// TwinCAT 3 PLC project Xts_Library
// Title: Xts Library
// Company: BeckhoffUK
// Author: ChrisK
// ProjectVersion: 7.2.0.0
// Description: Xts framework implementation
// ProgramVersion: 3.1.4026.13
// libraries:
//   Base Library, * (Beckhoff UK)
//   Motion Library, * (Beckhoff UK)
//   Tc2_MC2, * (Beckhoff Automation GmbH)
//   Tc2_Standard, * (Beckhoff Automation GmbH)
//   Tc2_System, * (Beckhoff Automation GmbH)
//   Tc3_Mc3Definitions, * (Beckhoff Automation GmbH)
//   Tc3_McCollisionAvoidance, * (Beckhoff Automation GmbH)
//   Tc3_McCoordinatedMotion, * (Beckhoff Automation GmbH)
//   Tc3_Module, * (Beckhoff Automation GmbH)
//   Tc3_PackML_V2, * (Beckhoff Automation GmbH)
//   Tc3_XTS_Utility, * (Beckhoff Automation GmbH)
// project tree:
//   Mover Class/ ITF_XtsMoverAxis.TcIO, XtsMoverAxis.TcPOU
//   SequenceSamples/ IndexMoverSequence.TcPOU, IndexSequenceState.TcDUT, MoverSequenceInfo.TcDUT
//   Station Class/Process/ IProcess.TcIO, Process.TcPOU
//   Station Class/Station/ IStation.TcIO, Station.TcPOU, StationSample.TcPOU, stStationInfo.TcDUT, stStationStatus.TcDUT
//   Station Class/TMSStation/ ITF_SwitchStation.TcIO, TmsEmbarkSingleSwitch.TcPOU, TmsEmbarkStation.TcPOU, TmsHoldStation.TcPOU
//   / SystemParameters.TcGVL
//   Tasks/ ActivateTrackForMover.TcPOU, AddMoverToGroupTask.TcPOU, DisableGroup.TcPOU, EnableGroup.TcPOU, GearInCA.TcPOU, HaltMover.TcPOU, MoveModuloMoverToPosition.TcPOU, RemoveAllMoverFromGroup.TcPOU, RemoveMoverFromGroup.TcPOU, ResetGroup.TcPOU, StopMoverGroup.TcPOU, XtsDisableSequence.TcPOU, XtsEnableSequence.TcPOU
//   XTS Class/XPU/ ITF_XTSIOEnvVarWrapper.TcIO, XTSIOEnvVarWrapper.TcPOU
//   XTS Class/Xts Collision Group/ CAGroupInfo.TcDUT, CAGroupStatus.TcDUT, CollisionGroup.TcPOU, ICollisionGroup.TcIO, ITF_CAMover.TcIO
//   XTS Class/Xts Hardware/ I_XtsTrack.TcIO, XtsSystemInitialisation.TcDUT, XTSHardware_V2.TcPOU, XtsMotorModule.TcPOU, XtsPart.TcPOU, XtsTrack.TcPOU
//   XTS Class/ Xts.TcPOU
// real-time tasks:
//   TASK PlcTask: cycle T#10ms, priority 20, ADS port 350

// ---- SequenceSamples/IndexSequenceState.TcDUT
{attribute 'qualified_only'}
{attribute 'strict'}
TYPE IndexSequenceState :
(
	Init := 0,                                               
	Available := 1,
	MovingToStart := 2, 
	AtStart := 3,                                 
	MovingToStation := 4,
	QueuedAtStation := 5,
	AtStation := 6,
	AtProcess := 7,
	InProcess := 8,
	GetNextMove := 9,
	GoToNextStation := 10,
	Stopping := 11,
	Aborting := 12
);
END_TYPE

// ---- SequenceSamples/MoverSequenceInfo.TcDUT
TYPE MoverSequenceInfo :
STRUCT
	MoverId : UDINT;
	CurrentStation : INT;
	Velocity : MC_LREAL;
	State : IndexSequenceState;
END_STRUCT
END_TYPE

// ---- Station Class/Station/stStationInfo.TcDUT
TYPE stStationInfo :
STRUCT
	StationProcessTime : TIME;
	StationPosition : MC_LREAL;
	StationStatus : stStationStatus;
END_STRUCT
END_TYPE

// ---- Station Class/Station/stStationStatus.TcDUT
TYPE stStationStatus :
STRUCT
	Empty : BOOL;
	Complete : BOOL;
	Operating : BOOL;
	Ready : BOOL;
	HasMover : BOOL;
END_STRUCT
END_TYPE

// ---- XTS Class/Xts Collision Group/CAGroupInfo.TcDUT
TYPE CAGroupInfo :
STRUCT
	sName 		: STRING;
	nId			: OTCID;
	eGroupState	: MC_GROUP_STATE;
	nAxesCount 	: INT; 
END_STRUCT
END_TYPE

// ---- XTS Class/Xts Collision Group/CAGroupStatus.TcDUT
{attribute 'qualified_only'}
{attribute 'strict'}
TYPE CAGroupStatus :
(
	mcGroupStateInvalid:=0, 
	mcGroupStateDisabled:=1,
	mcGroupStateStandby:=2, 
	mcGroupStateMoving:=3, 
	mcGroupStateStopping:=4, 
	mcGroupStateErrorStop:=5, 
	mcGroupStateHoming:=6, 
	mcGroupStateNotReady:=7, 
	mcGroupAllAxesStanding:=8,
    mcGroupConstantVelocity:=9,
    mcGroupAccelerating:=10,
    mcGroupDecelerating:=11,
    mcGroupInPosition:=12,
    mcGroupError:=13
);
END_TYPE

// ---- XTS Class/Xts Hardware/XtsSystemInitialisation.TcDUT
{attribute 'qualified_only'}
{attribute 'strict'}
TYPE XtsSystemInitialisation :
(
	Init := 0,
	PassGroupReference := 1,
	InitialiseHardware := 2,
	SetDetection := 3,                                              
	Redetect := 4,
	MoversValid := 5,                                 
	AllMoversFound := 6,
	MoverIdDetection := 7,
	XTSMode := 8,
	CheckModuleVoltages := 9,
	HWReady := 10,
	HWError := 999
);
END_TYPE

// ---- SystemParameters.TcGVL
{attribute 'qualified_only'}
VAR_GLOBAL CONSTANT
	MaxModulesInPart  : UINT := 20;
	MaxPartsInTrack : UINT := 5;
	NumberOfMovers : UINT := 10;
	NumberOfStations : UINT := 6;
	NumberOfParts : UINT := 1;
	NumberOfTracks : UINT := 2;
END_VAR

// ---- Mover Class/ITF_XtsMoverAxis.TcIO
INTERFACE ITF_XtsMoverAxis

PROPERTY Acceleration : mc_lreal
GET
END_GET
SET
END_SET
END_PROPERTY

METHOD ActivateTrack : HRESULT
VAR_INPUT
	NewTrack : OTCID;
	Track : I_XtsTrack;
END_VAR
END_METHOD

PROPERTY AxisRef : Reference to Axis_ref
GET
END_GET
END_PROPERTY

PROPERTY Deceleration : mc_lreal
GET
END_GET
SET
END_SET
END_PROPERTY

METHOD DisableMover : HRESULT
VAR_INPUT
END_VAR
END_METHOD

METHOD EnableMover : HRESULT
VAR_INPUT
END_VAR
END_METHOD

PROPERTY Gap : MC_LREAL
GET
END_GET
SET
END_SET
END_PROPERTY

METHOD PUBLIC Gear : HRESULT
VAR_INPUT
	MasterPosition : MC_LREAL;
	SlavePosition : MC_LREAL;
END_VAR
END_METHOD

METHOD HaltAxis : HRESULT
VAR_INPUT
END_VAR
END_METHOD

PROPERTY PUBLIC IdentInGroup : IDENT_IN_GROUP_REF
GET
END_GET
END_PROPERTY

METHOD isMoverAtPosition : BOOL
VAR_INPUT
	Position : MC_LREAL;
END_VAR
END_METHOD

METHOD isMoverDetected : BOOL
VAR_INPUT
END_VAR
END_METHOD

METHOD isMoverEnabled : BOOL
VAR_INPUT
END_VAR
END_METHOD

METHOD isMoverStationary : BOOL
VAR_INPUT
END_VAR
END_METHOD

PROPERTY Jerk : mc_lreal
GET
END_GET
SET
END_SET
END_PROPERTY

PROPERTY PUBLIC MoverErrorID : DWORD
GET
END_GET
END_PROPERTY

PROPERTY PUBLIC MoversActiveTrack : OTCID
GET
END_GET
END_PROPERTY

PROPERTY PUBLIC MoverXtsIoEnvInterface : I_TcIoXtsXpuMover
GET
END_GET
SET
END_SET
END_PROPERTY

METHOD MoveTo : HRESULT
VAR_INPUT
	RequiredPosition : MC_LREAL;
	MoveVelocity : MC_LREAL;
	NonModuloMove : BOOL;
END_VAR
END_METHOD

PROPERTY MyCAGroup : ITF_CAMover
GET
END_GET
SET
END_SET
END_PROPERTY

PROPERTY MyMasterRef : REFERENCE TO AXIS_REF
GET
END_GET
SET
END_SET
END_PROPERTY

PROPERTY PositiveDirectionOnly : BOOL
GET
END_GET
SET
END_SET
END_PROPERTY

METHOD ResetAxis : HRESULT
VAR_INPUT
END_VAR
END_METHOD

METHOD TriggerMoverArrive : BOOL
VAR_INPUT
END_VAR
END_METHOD

METHOD TriggerMoverLeave : BOOL
VAR_INPUT
END_VAR
END_METHOD

END_INTERFACE

// ---- Station Class/Process/IProcess.TcIO
INTERFACE IProcess EXTENDS IStation

PROPERTY EndPosition : MC_LREAL
GET
END_GET
SET
END_SET
END_PROPERTY

PROPERTY IsProcess : booL
GET
END_GET
SET
END_SET
END_PROPERTY

PROPERTY ProcessVelocity : mc_lreal
GET
END_GET
SET
END_SET
END_PROPERTY

PROPERTY StartPosition : MC_LREAL
GET
END_GET
SET
END_SET
END_PROPERTY

END_INTERFACE

// ---- Station Class/Station/IStation.TcIO
INTERFACE IStation

METHOD Abort : BOOL
VAR_INPUT
END_VAR
END_METHOD

METHOD HasMover : BOOL
VAR_INPUT
	mover : ITF_XtsMoverAxis;
END_VAR
END_METHOD

METHOD IsClear : BOOL
VAR_INPUT
END_VAR
END_METHOD

METHOD isComplete : BOOL
VAR_INPUT
END_VAR
END_METHOD

PROPERTY IsLastStation : BOOL
GET
END_GET
SET
END_SET
END_PROPERTY

METHOD IsOperating : BOOL
VAR_INPUT
END_VAR
END_METHOD

METHOD IsReady : BOOL
VAR_INPUT
END_VAR
END_METHOD

METHOD MoverAway : BOOL
VAR_INPUT
END_VAR
END_METHOD

PROPERTY Position : MC_LREAL
GET
END_GET
SET
END_SET
END_PROPERTY

END_INTERFACE

// ---- Station Class/TMSStation/ITF_SwitchStation.TcIO
INTERFACE ITF_SwitchStation EXTENDS __SYSTEM.IQueryInterface

METHOD SwitchMoveComplete : BOOL
VAR_INPUT
END_VAR
END_METHOD

END_INTERFACE

// ---- XTS Class/XPU/ITF_XTSIOEnvVarWrapper.TcIO
INTERFACE ITF_XTSIOEnvVarWrapper

METHOD GetCaGroupInterface : I_Mc2CaGroup
VAR_INPUT
	CAGroupNumber : INT;
END_VAR
END_METHOD

METHOD PUBLIC GetMotorModuleInterface : I_TcIoXtsPartModule
VAR_INPUT
	PartNumber : INT;
	ModuleNumber : INT;
END_VAR
END_METHOD

METHOD PUBLIC GetMoverInterface : I_TcIoXtsXpuMover
VAR_INPUT
	MoverId : INT;
END_VAR
END_METHOD

METHOD PUBLIC GetPartInterface : I_TcIoXtsXpuPart
VAR_INPUT
	PartNumber : INT;
END_VAR
END_METHOD

METHOD PUBLIC GetTrackInterface : I_TcIoXtsXpuTrack
VAR_INPUT
	TrackNumber : INT;
END_VAR
END_METHOD

METHOD GetXPUInterface : I_TcIoXtsProcessingUnit
VAR_INPUT
END_VAR
END_METHOD

METHOD IsInitialised : BOOL
VAR_INPUT
END_VAR
END_METHOD

METHOD IsInSim : BOOL
VAR_INPUT
END_VAR
END_METHOD

END_INTERFACE

// ---- XTS Class/Xts Collision Group/ICollisionGroup.TcIO
INTERFACE ICollisionGroup

METHOD AddMoverToThisGroup : HRESULT
VAR_INPUT
	MoverToAdd : ITF_XtsMoverAxis;
END_VAR
END_METHOD

METHOD Disable : BOOL
VAR_INPUT
END_VAR
END_METHOD

METHOD Enable : BOOL
VAR_INPUT
END_VAR
END_METHOD

METHOD GetAxisCount : udint
VAR_INPUT
END_VAR
END_METHOD

PROPERTY GroupRef : reference to AXES_GROUP_REF
GET
END_GET
END_PROPERTY

PROPERTY GroupState : CAGroupStatus
GET
END_GET
END_PROPERTY

METHOD GroupStop : HRESULT
VAR_INPUT
END_VAR
END_METHOD

METHOD RemoveAllMovers : HRESULT
VAR_INPUT
END_VAR
END_METHOD

METHOD Reset : BOOL
VAR_INPUT
END_VAR
END_METHOD

END_INTERFACE

// ---- XTS Class/Xts Collision Group/ITF_CAMover.TcIO
INTERFACE ITF_CAMover

METHOD AddMoverToThisGroup : HRESULT
VAR_INPUT
	MoverToAdd : ITF_XtsMoverAxis;
END_VAR
END_METHOD

METHOD RemoveAMover : BOOL
VAR_INPUT
	moverId : UDINT;
END_VAR
END_METHOD

END_INTERFACE

// ---- XTS Class/Xts Hardware/I_XtsTrack.TcIO
INTERFACE I_XtsTrack

PROPERTY MyOTCID : OTCID
GET
END_GET
SET
END_SET
END_PROPERTY

PROPERTY TrackLength : MC_Lreal
GET
END_GET
END_PROPERTY

END_INTERFACE

// ---- Mover Class/XtsMoverAxis.TcPOU
FUNCTION_BLOCK XtsMoverAxis EXTENDS CyclicBase IMPLEMENTS ITF_XtsMoverAxis
VAR
	MyAxisRef : AXIS_REF;
	_MyAxisStatus : ST_AxisStatus;
	_MyNCData : NCTOPLC_AXIS_REF;
	MoverPowerCommand : AxisPower(MyAxisRef);
	MoverMoveCommand : MoveModuloMoverToPosition(MyAxisRef) := (Gap := 100.0);
	MoverHaltCommand : HaltMover(MyAxisRef);
	MoverResetCommand : AxesReset(MyAxisRef);
	MoverActivateTrackCommand : ActivateTrackForMover(MyAxisRef);
	axesGear	: GearInCA(MyAxisRef);
	_ipTcIoXtsMover	: I_TcIoXtsXpuMover;
	_ActiveTrackLength : MC_LREAL;
	TrackChangeTrigger : R_TRIG;
	_MoverAbsMoveOptions : ST_MoveAbsoluteCAOptions;
	_stTmsActPositions			: ST_PositionInfo;
	_CurrentTrack : I_XtsTrack;
	_MyCAGroup : ITF_CAMover;
	_ForwardOnly : BOOL := TRUE;
END_VAR
VAR CONSTANT
	_MaxMoverVelocity : MC_LREAL := 4000.0;
END_VAR

PROPERTY PUBLIC Acceleration : MC_LREAL
GET
Acceleration := MoverMoveCommand.Acceleration;
END_GET
SET
MoverMoveCommand.Acceleration := Acceleration;
END_SET
END_PROPERTY

METHOD ActivateTrack : HRESULT
VAR_INPUT
	NewTrack : OTCID;
	Track : I_XtsTrack;
END_VAR
IF NOT MoverActivateTrackCommand.Busy AND THIS^.isMoverStationary() AND NewTrack <> 0  THEN
	IF MoverActivateTrackCommand.Execute(Track := Track.MyOTCID) THEN
		_CurrentTrack := Track;
		_ActiveTrackLength := Track.TrackLength;
		ActivateTrack := 1;
	ELSE
		ActivateTrack := -1;
	END_IF
ELSE
	ActivateTrack := -1;
END_IF
END_METHOD

METHOD ActivateZeroReferenceSystem : HRESULT
VAR_INPUT
	NewTrack : OTCID;
END_VAR
IF NOT MoverActivateTrackCommand.Busy AND THIS^.isMoverStationary() THEN // AND NewTrack <> 0  THEN
	IF MoverActivateTrackCommand.Execute(Track := NewTrack) THEN
		_CurrentTrack := 0;
		ActivateZeroReferenceSystem := 1;
	ELSE
		ActivateZeroReferenceSystem := -1;
	END_IF
ELSE
	ActivateZeroReferenceSystem := -1;
END_IF
END_METHOD

PROPERTY AxisRef : Reference to Axis_ref
GET
AxisRef REF= MyAxisRef;
END_GET
END_PROPERTY

METHOD PUBLIC  Cycle : HRESULT
VAR_INPUT
END_VAR
IF isMoverDetected() THEN
	MoverPowerCommand.Cycle();
	MoverMoveCommand.Cycle();
	MoverHaltCommand.Cycle();
	MoverResetCommand.Cycle();
	MoverActivateTrackCommand.Cycle();
	axesGear.Cycle();
	TrackChangeTrigger(CLK := MoverActivateTrackCommand.Done);
	IF TrackChangeTrigger.Q THEN
		_MoverAbsMoveOptions.PositionReferenceSystem :=  MoverActivateTrackCommand.NewTrackId;
		_MoverAbsMoveOptions.DynamicsReferenceSystem := MoverActivateTrackCommand.NewTrackId;
		MoverMoveCommand.Options := _MoverAbsMoveOptions;	
	END_IF
	IF _ipTcIoXtsMover <> 0 THEN
		_stTmsActPositions := _ipTcIoXtsMover.GetPositionInfo();
	END_IF
	Cycle := 1;
ELSE
	Cycle := -1;
END_IF
MyAxisRef.ReadStatus();
_MyNCData := MyAxisRef.NcToPlc;
_MyAxisStatus := MyAxisRef.Status;
END_METHOD

PROPERTY PUBLIC Deceleration : MC_LREAL
GET
Deceleration := MoverMoveCommand.Deceleration;
END_GET
SET
MoverMoveCommand.Deceleration := Deceleration;
MoverHaltCommand.Deceleration := Deceleration;
END_SET
END_PROPERTY

METHOD PUBLIC DisableMover : HRESULT
VAR_INPUT
END_VAR
IF THIS^.isMoverEnabled() AND NOT MoverPowerCommand.Busy THEN
	MoverPowerCommand.Disable();
	DisableMover := 1;
ELSE
	DisableMover := -1;
END_IF
END_METHOD

METHOD PUBLIC EnableMover : HRESULT
VAR_INPUT
END_VAR
IF (NOT MoverPowerCommand.Busy) AND NOT THIS^.isMoverEnabled() THEN // AND _CurrentTrack <> 0 THEN
	MoverPowerCommand.Enable();
	EnableMover := 1;
ELSE
	EnableMover := -1;
END_IF
END_METHOD

PROPERTY PUBLIC Gap : MC_LREAL
GET
Gap := MoverMoveCommand.Gap;
END_GET
SET
IF Gap >= 50.0 THEN
	MoverMoveCommand.Gap := Gap;
	MoverHaltCommand.Gap := Gap;
ELSE
	Gap := 100.0;
END_IF
END_SET
END_PROPERTY

METHOD PUBLIC Gear : HRESULT
VAR_INPUT
	MasterPosition : MC_LREAL;
	SlavePosition : MC_LREAL;
END_VAR
IF NOT axesGear.Busy AND __ISVALIDREF(axesGear.MyGearMaster) AND MasterPosition <= _ActiveTrackLength AND SlavePosition <= _ActiveTrackLength THEN
	IF axesGear.Sync(MasterPosition := MasterPosition, SlavePosition := SlavePosition) THEN
		Gear := 1;
	ELSE
		Gear := -1;
	END_IF
ELSE
	Gear := -1;
END_IF
END_METHOD

METHOD GetMoverCtrlOTCID : XtsMoverControllerOTCID
VAR_INPUT
END_VAR
GetMoverCtrlOTCID := _ipTcIoXtsMover.P_MoverControllerOid;
END_METHOD

METHOD GetMoverOTCID : OTCID
VAR_INPUT
END_VAR
//GetMoverCtrlOTCID := _ipTcIoXtsMover.P_AxisOid;
END_METHOD

METHOD PUBLIC HaltAxis : HRESULT
VAR_INPUT
END_VAR
IF NOT MoverHaltCommand.Busy THEN// AND NOT THIS^.isMoverStationary() THEN
	IF MoverHaltCommand.Execute() THEN
		HaltAxis := 1;
	ELSE
		HaltAxis := -1;
	END_IF
ELSE
	HaltAxis := -1;
END_IF
END_METHOD

PROPERTY PUBLIC IdentInGroup : IDENT_IN_GROUP_REF
GET
IdentInGroup := UDINT_TO_IDENTINGROUP(id := _MyNCData.AxisId);
END_GET
END_PROPERTY

METHOD inGear : BOOL
VAR_INPUT
END_VAR
inGear := axesGear.GearInPosCA.InSync;
END_METHOD

METHOD IsActive : BOOL
VAR_INPUT
END_VAR
IsActive := _ipTcIoXtsMover.GetIsActive();
END_METHOD

METHOD PUBLIC isMoverAtPosition : BOOL
VAR_INPUT
	Position : MC_LREAL;
END_VAR
IF Position > 1 THEN
	IF _stTmsActPositions.fTrackPosition < position + 1 AND _stTmsActPositions.fTrackPosition > position - 1 THEN
		isMoverAtPosition := TRUE;
	ELSE
		isMoverAtPosition := FALSE;
	END_IF  
ELSE
	IF _stTmsActPositions.fTrackPosition < position + 1 AND _stTmsActPositions.fTrackPosition > 0.0  
		OR _stTmsActPositions.fTrackPosition < _CurrentTrack.TrackLength AND _stTmsActPositions.fTrackPosition > _CurrentTrack.TrackLength - 1 THEN
		isMoverAtPosition := TRUE;
	ELSE
		isMoverAtPosition := FALSE;
	END_IF
END_IF
END_METHOD

METHOD PUBLIC isMoverDetected : BOOL
VAR_INPUT
END_VAR
isMoverDetected := _MyNCData.AxisId <> 0;
END_METHOD

METHOD PUBLIC isMoverEnabled : BOOL
VAR_INPUT
END_VAR
isMoverEnabled :=  NOT _MyAxisStatus.Disabled;
END_METHOD

METHOD PUBLIC isMoverStationary : BOOL
VAR_INPUT
END_VAR
isMoverStationary := _MyAxisStatus.NotMoving;
END_METHOD

PROPERTY PUBLIC Jerk : MC_LREAL
GET
Jerk := MoverMoveCommand.Jerk;
END_GET
SET
MoverMoveCommand.Jerk := Jerk;
MoverHaltCommand.Jerk := Jerk;
END_SET
END_PROPERTY

PROPERTY PUBLIC MoverErrorID : DWORD
GET
MoverErrorID := _MyAxisStatus.ErrorID;
END_GET
END_PROPERTY

PROPERTY PUBLIC MoversActiveTrack : OTCID
GET
MoversActiveTrack := _ipTcIoXtsMover.GetActiveTrackObjectId();
END_GET
END_PROPERTY

PROPERTY PUBLIC MoverXtsIoEnvInterface : I_TcIoXtsXpuMover
GET
MoverXtsIoEnvInterface := _ipTcIoXtsMover;
END_GET
SET
_ipTcIoXtsMover := MoverXtsIoEnvInterface;
END_SET
END_PROPERTY

METHOD PUBLIC MoveTo : HRESULT
VAR_INPUT
	RequiredPosition : MC_LREAL;
	MoveVelocity : MC_LREAL;
	NonModuloMove : BOOL;
END_VAR
IF NOT MoverMoveCommand.Busy AND MoveVelocity < _MaxMoverVelocity AND (*RequiredPosition < _ActiveTrackLength AND*) Gap >= 50.0 THEN
	IF NonModuloMove THEN
		IF THIS^.MoverMoveCommand.MoveTo(Position := RequiredPosition, 
										Velocity := MoveVelocity, 
										Direction := Tc3_Mc3Definitions.MC_DIRECTION.mcDirectionNonModulo, 
										Turns := 0) THEN
										
			MoveTo := 1;
		END_IF
	ELSE
		IF _ForwardOnly THEN
			THIS^.MoverMoveCommand.MoveTo(Position := RequiredPosition, 
										Velocity := MoveVelocity, 
										Direction := Tc3_Mc3Definitions.MC_DIRECTION.mcDirectionPositive, 
										Turns := 0);
			MoveTo := 1;
		ELSE
			IF RequiredPosition > MyAxisRef.NcToPlc.ModuloActPos THEN
				IF THIS^.MoverMoveCommand.MoveTo(Position := RequiredPosition, 
											Velocity := MoveVelocity, 
											Direction := Tc3_Mc3Definitions.MC_DIRECTION.mcDirectionPositive, 
											Turns := 0) THEN
											
					MoveTo := 1;
				END_IF
			ELSE
				IF THIS^.MoverMoveCommand.MoveTo(Position := RequiredPosition, 
											Velocity := MoveVelocity, 
											Direction := Tc3_Mc3Definitions.MC_DIRECTION.mcDirectionNegative, 
											Turns := 0) THEN
											
					MoveTo := 1;
				END_IF	
			END_IF
		END_IF
	END_IF
ELSE
	MoveTo := -1;
END_IF
END_METHOD

PROPERTY MyCAGroup : ITF_CAMover
GET
MyCAGroup := _MyCAGroup;
END_GET
SET
_MyCAGroup := MyCAGroup;
END_SET
END_PROPERTY

PROPERTY MyMasterRef : REFERENCE TO AXIS_REF
GET
MyMasterRef REF= axesGear.MyGearMaster;
END_GET
SET
axesGear.MyGearMaster REF= MyMasterRef;
END_SET
END_PROPERTY

PROPERTY PositiveDirectionOnly : BOOL
GET
PositiveDirectionOnly := _ForwardOnly;
END_GET
SET
_ForwardOnly := PositiveDirectionOnly;
END_SET
END_PROPERTY

METHOD PUBLIC ResetAxis : HRESULT
VAR_INPUT
END_VAR
IF NOT MoverResetCommand.Busy AND _MyAxisStatus.Error THEN
	IF MoverResetCommand.Execute() = S_OK THEN
		ResetAxis := 1;
	ELSE
		ResetAxis := -1;
	END_IF
ELSE
	ResetAxis := -1;
END_IF
END_METHOD

METHOD SetForceCouple : HRESULT
VAR_INPUT
	XtsMoverCtrlOTCID : Tc3_XTS_Utility.XtsMoverControllerOTCID;
END_VAR
_ipTcIoXtsMover.MoverController.SetForceCouple(nForceCouple := XtsMoverCtrlOTCID);
END_METHOD

METHOD SwapMover : HRESULT
VAR_INPUT
    MoverToSwapWith : MoverOTCID;
END_VAR
_ipTcIoXtsMover.swapmover(nSwapMoverObjectId := MoverToSwapWith);
END_METHOD

METHOD TriggerMoverArrive : BOOL
VAR_INPUT
END_VAR
_ipTcIoXtsMover.TriggerArrive();
END_METHOD

METHOD TriggerMoverLeave : BOOL
VAR_INPUT
END_VAR
TriggerMoverLeave := _ipTcIoXtsMover.TriggerLeave();
END_METHOD

END_FUNCTION_BLOCK

// ---- Tasks/MoveModuloMoverToPosition.TcPOU
FUNCTION_BLOCK MoveModuloMoverToPosition EXTENDS TaskBase
VAR_INPUT
END_VAR
VAR_OUTPUT
END_VAR
VAR
	moveAbs	: MC_MoveAbsoluteCA;
	_Axis : REFERENCE TO AXIS_REF;
	_MoveMover : BOOL;
	_stOptions : ST_MoveAbsoluteCAOptions;
	_ErrorId: UDINT;
END_VAR

{analysis -2}

METHOD Abort : BOOL
moveAbs.Execute := FALSE;
moveAbs.Position := moveAbs.Velocity := 0;
_MoveMover := false;
_Busy := FALSE;
Abort := true;
State := 0;
END_METHOD

PROPERTY PUBLIC Acceleration : mc_lreal
GET
Acceleration := moveAbs.Acceleration;
END_GET
SET
moveAbs.Acceleration := Acceleration;
END_SET
END_PROPERTY

METHOD Cycle : HRESULT
VAR_INPUT
END_VAR
Cycle := S_OK;
CASE State OF
	0:
		IF _MoveMover THEN
			Cycle := S_PENDING;
			_Done := FALSE;
			_Error := FALSE;
			_Busy := TRUE;
			moveAbs.Execute := TRUE;
			IF moveAbs.Busy THEN
				State := 10;
				_MoveMover := FALSE;
			END_IF
		END_IF
		
	10:
		IF NOT moveAbs.Busy THEN
			IF moveAbs.Done THEN
				_Done := TRUE;
			ELSIF moveAbs.Error THEN
				_Error := TRUE;
				_ErrorId := moveAbs.ErrorId;
			END_IF
			_Busy := FALSE;
			moveAbs.Execute := FALSE;
			State := 0;
			Cycle := S_OK;
		END_IF
	ELSE
		Cycle := E_FAIL;
END_CASE

moveAbs(Axis := _Axis, Options := _stOptions);
END_METHOD

PROPERTY PUBLIC Deceleration : mc_lreal
GET
Deceleration := moveAbs.Deceleration;
END_GET
SET
moveAbs.Deceleration := Deceleration;
END_SET
END_PROPERTY

METHOD FB_init : BOOL
VAR_INPUT
	bInitRetains : BOOL; // if TRUE, the retain variables are initialized (warm start / cold start)
	bInCopyCode : BOOL;  // if TRUE, the instance afterwards gets moved into the copy code (online change)
	axis : reference TO AXIS_REF;
END_VAR
_Axis REF= axis;
END_METHOD

PROPERTY PUBLIC Gap : mc_lreal
GET
Gap := moveAbs.Gap;
END_GET
SET
moveAbs.Gap := Gap;
END_SET
END_PROPERTY

PROPERTY PUBLIC Jerk : mc_lreal
GET
Jerk := moveAbs.Jerk;
END_GET
SET
moveAbs.Jerk := Jerk;
END_SET
END_PROPERTY

METHOD MoveTo : BOOL
VAR_INPUT
	Position : MC_LREAL;
	Velocity : MC_LREAL;
	Direction: Tc3_Mc3Definitions.MC_DIRECTION;
	Turns: UDINT;
END_VAR
moveAbs.Position := Position;
moveAbs.Velocity := Velocity;
moveAbs.Direction := Direction;
moveAbs.Options.AdditionalTurns := Turns;
_MoveMover := MoveTo := true;
END_METHOD

PROPERTY PUBLIC Options : ST_MoveAbsoluteCAOptions
GET
Options := _stOptions;
END_GET
SET
_stOptions := Options;
END_SET
END_PROPERTY

END_FUNCTION_BLOCK

// ---- Tasks/HaltMover.TcPOU
FUNCTION_BLOCK HaltMover EXTENDS TaskBase
VAR_INPUT
END_VAR
VAR_OUTPUT
END_VAR
VAR
	haltMoverCA : Tc3_McCollisionAvoidance.MC_HaltCA;
	_Axis : REFERENCE TO Tc2_MC2.AXIS_REF;
	_HaltMover : BOOL;
END_VAR

{analysis -2}

METHOD Abort : BOOL
haltMoverCA.Execute := FALSE;
_Busy := FALSE;
_HaltMover := FALSE;
Abort := TRUE;
State := 0;
END_METHOD

METHOD Cycle : HRESULT
VAR_INPUT
END_VAR
Cycle := S_OK;
CASE State OF
	0:
		IF _HaltMover THEN
			Cycle := S_PENDING;
			_Done := FALSE;
			_Error := FALSE;
			_Busy := TRUE;
			haltMoverCA.Execute := TRUE;
			IF haltMoverCA.Busy THEN
				State := 10;
				_HaltMover := FALSE;
			END_IF
		END_IF
	
	10:
		IF NOT haltMoverCA.Busy THEN
			IF haltMoverCA.Done THEN
				_Done := TRUE;
			ELSIF haltMoverCA.Error THEN
				_Error := TRUE;
			END_IF
			_Busy := FALSE;
			haltMoverCA.Execute := FALSE;
			State := 0;
			Cycle := S_OK;
		END_IF
	ELSE
		Cycle := E_FAIL;
END_CASE

haltMoverCA(Axis := _Axis);
END_METHOD

PROPERTY Deceleration : MC_LREAL
GET
Deceleration := haltMoverCA.Deceleration;
END_GET
SET
haltMoverCA.Deceleration := Deceleration;
END_SET
END_PROPERTY

METHOD Execute : BOOL
VAR_INPUT
END_VAR
IF NOT _HaltMover THEN
	Execute := _HaltMover := TRUE;
ELSE
	Execute := false;
END_IF
END_METHOD

METHOD FB_init : BOOL
VAR_INPUT
	bInitRetains : BOOL; // if TRUE, the retain variables are initialized (warm start / cold start)
	bInCopyCode : BOOL;  // if TRUE, the instance afterwards gets moved into the copy code (online change)
	Axis : reference TO AXIS_REF;
END_VAR
_Axis REF= Axis;
END_METHOD

PROPERTY Gap : MC_LREAL
GET
Gap := haltMoverCA.Gap;
END_GET
SET
haltMoverCA.Gap := Gap;
END_SET
END_PROPERTY

PROPERTY Jerk : MC_LREAL
GET
Jerk := haltMoverCA.Jerk;
END_GET
SET
haltMoverCA.Jerk := Jerk;
END_SET
END_PROPERTY

END_FUNCTION_BLOCK

// ---- Tasks/ActivateTrackForMover.TcPOU
FUNCTION_BLOCK ActivateTrackForMover EXTENDS TaskBase
VAR_INPUT
END_VAR
VAR_OUTPUT
END_VAR
VAR
	mcActivateTrack : Tc3_McCollisionAvoidance.MC_ActivateTrack;
	_Axis : REFERENCE TO Tc2_MC2.AXIS_REF;
	_ActivateTrack : BOOL;
	_newTrackId : OTCID;
	_errorId: UDINT;
END_VAR

{analysis -2}

METHOD Abort : BOOL
mcActivateTrack.Execute := FALSE;
_Busy := FALSE;
_ActivateTrack := FALSE;
Abort := TRUE;
State := 0;
END_METHOD

METHOD Cycle : HRESULT
VAR_INPUT
END_VAR
Cycle := S_OK;
CASE State OF
	0:
		IF _ActivateTrack THEN
			Cycle := S_PENDING;
			_Done := FALSE;
			_Error := FALSE;
			_Busy := TRUE;
			mcActivateTrack.Execute := TRUE;
			IF mcActivateTrack.Busy THEN
				State := 10;
				_ActivateTrack := FALSE;
			END_IF
		END_IF
	
	10:
		IF NOT mcActivateTrack.Busy THEN
			IF mcActivateTrack.Done THEN
				_Done := TRUE;
				_newTrackId := mcActivateTrack.TrackId;
			ELSIF mcActivateTrack.Error THEN
				_Error := TRUE;
				_errorId := mcActivateTrack.ErrorId;
			END_IF
			_Busy := FALSE;
			mcActivateTrack.Execute := FALSE;
			State := 0;
			Cycle := S_OK;
		END_IF
	ELSE
		Cycle := E_FAIL;
END_CASE

mcActivateTrack(Axis := _Axis);
END_METHOD

METHOD PUBLIC Execute : BOOL
VAR_INPUT
	Track : OTCID;
END_VAR
IF NOT _ActivateTrack THEN
	Execute := _ActivateTrack := TRUE;
	mcActivateTrack.TrackId := Track;
ELSE
	Execute := false;
END_IF;
END_METHOD

METHOD FB_init : BOOL
VAR_INPUT
	bInitRetains : BOOL; // if TRUE, the retain variables are initialized (warm start / cold start)
	bInCopyCode : BOOL;  // if TRUE, the instance afterwards gets moved into the copy code (online change)
	Axis : reference TO AXIS_REF;
END_VAR
_Axis REF= Axis;
END_METHOD

PROPERTY PUBLIC NewTrackId : OTCID
GET
NewTrackId := _newTrackId;
END_GET
END_PROPERTY

END_FUNCTION_BLOCK

// ---- Tasks/GearInCA.TcPOU
FUNCTION_BLOCK PUBLIC GearInCA EXTENDS TaskBase
VAR
	GearInPosCA : Tc3_McCollisionAvoidance.MC_GearInPosCA;
	_syncStrategy : Tc3_Mc3Definitions.MC_SYNC_STRATEGY := Tc3_Mc3Definitions.MC_SYNC_STRATEGY.mcSyncStrategyEarly;
	_SlaveAxis : REFERENCE TO Tc2_MC2.AXIS_REF;
	_MasterAxis : REFERENCE TO Tc2_MC2.AXIS_REF;
	_GearMover: BOOL;
	_ErrorID: UDINT;
END_VAR

{analysis -2}

METHOD Abort : BOOL
GearInPosCA.Execute := FALSE;
_GearMover := FALSE;
_Busy := false;
Abort := true;
State := 0;
END_METHOD

METHOD Cycle : HRESULT
VAR_INPUT
END_VAR
Cycle := S_OK;
CASE State OF
	0:
		IF _GearMover THEN
			Cycle := S_PENDING;
			_Done := FALSE;
			_Error := FALSE;
			_Busy := TRUE;
			GearInPosCA.Execute := TRUE;
			IF GearInPosCA.Busy THEN
				State := 10;
				_GearMover := FALSE;
			END_IF
		END_IF
		
	10:
		IF GearInPosCA.InSync THEN
			GearInPosCA.Execute := FALSE;
			_Busy := FALSE;
			_Done := TRUE;
			State := 0;
			Cycle := S_OK;
		END_IF
	ELSE
		Cycle := E_FAIL;
END_CASE
_Error := GearInPosCA.Error;
_ErrorID := GearInPosCA.ErrorId;
IF __ISVALIDREF(_MasterAxis) AND __ISVALIDREF(_SlaveAxis) THEN
	GearInPosCA(Master := _MasterAxis, Slave := _SlaveAxis, SyncStrategy := _syncStrategy, Velocity := 2000.0, RatioNumerator := 1, Gap := 60.0);
END_IF
END_METHOD

METHOD FB_init : BOOL
VAR_INPUT
	bInitRetains : BOOL; // if TRUE, the retain variables are initialized (warm start / cold start)
	bInCopyCode : BOOL;  // if TRUE, the instance afterwards gets moved into the copy code (online change)
	axis : reference TO AXIS_REF;
END_VAR
_SlaveAxis REF= axis;
END_METHOD

PROPERTY MyGearMaster : REFERENCE TO AXIS_REF
GET
MyGearMaster REF= _MasterAxis;
END_GET
SET
_MasterAxis REF= MyGearMaster;
END_SET
END_PROPERTY

METHOD PUBLIC Sync : BOOL
VAR_INPUT
	MasterPosition : MC_LREAL;
	SlavePosition : MC_LREAL;
END_VAR
GearInPosCA.MasterSyncPosition := MasterPosition;
GearInPosCA.SlaveSyncPosition := SlavePosition;
_GearMover := Sync := true;
END_METHOD

PROPERTY PUBLIC SyncStrategy : mc_sync_strategy
GET
SyncStrategy := _syncStrategy;
END_GET
SET
_syncStrategy := SyncStrategy;
END_SET
END_PROPERTY

END_FUNCTION_BLOCK

// ---- SequenceSamples/IndexMoverSequence.TcPOU
FUNCTION_BLOCK IndexMoverSequence EXTENDS CyclicBase
VAR
	State : IndexSequenceState;  
	CurrentStation : UINT;
	TargetStationPosition : MC_LREAL;
	_MoverVelocity : MC_LREAL := 1000.0;
	stSequenceInfo : MoverSequenceInfo;
	StationArray : ARRAY[1..SystemParameters.NumberOfStations] OF IProcess;
	ThisMover : ITF_XtsMoverAxis;
	ExecuteSequence : BOOL;
	_startPosition : MC_LREAL;
	_XtsNoHome : BOOL;
	_NonModuloMoves : BOOL := false;
END_VAR

{analysis -2}

METHOD Abort : BOOL
VAR_INPUT
END_VAR
State := IndexSequenceState.Available;
CurrentStation := 0;
TargetStationPosition := 0.0;
stSequenceInfo.CurrentStation := UINT_TO_INT(CurrentStation);
stSequenceInfo.MoverId := ThisMover.AxisRef.NcToPlc.AxisId;
stSequenceInfo.State := State;
stSequenceInfo.Velocity := ThisMover.AxisRef.NcToPlc.ActVelo;
Abort := TRUE;
END_METHOD

METHOD PUBLIC  Cycle : HRESULT
VAR_INPUT
END_VAR
Cycle := S_OK;
CASE State OF
	IndexSequenceState.Init:
		IF ThisMover.isMoverDetected() THEN
			State := IndexSequenceState.Available;
		END_IF
		
	IndexSequenceState.Available:
		IF ExecuteSequence THEN
			State := IndexSequenceState.MovingToStart;
		END_IF
		
	IndexSequenceState.MovingToStart:
		IF ThisMover.isMoverAtPosition(position := _startPosition) OR _XtsNoHome THEN
			State := IndexSequenceState.AtStart;
		END_IF
			
	IndexSequenceState.AtStart:
		IF StationArray[1].IsReady() THEN
			State := IndexSequenceState.GetNextMove;
		END_IF

	IndexSequenceState.MovingToStation:
		IF ThisMover.isMoverStationary() THEN 
			IF ThisMover.isMoverAtPosition(TargetStationPosition) THEN
				IF StationArray[CurrentStation].IsProcess THEN
					State := IndexSequenceState.AtProcess;
				ELSE
					State := IndexSequenceState.AtStation;
				END_IF
				StationArray[CurrentStation].HasMover(ThisMover);
			ELSE
				State := IndexSequenceState.QueuedAtStation;
			END_IF
		END_IF
		
	IndexSequenceState.QueuedAtStation:
		IF NOT ThisMover.isMoverStationary() THEN
				State := IndexSequenceState.MovingToStation;
		END_IF

	IndexSequenceState.AtStation:
		IF StationArray[CurrentStation].isComplete() THEN
			State := IndexSequenceState.GetNextMove;
		END_IF

	IndexSequenceState.AtProcess:
		ThisMover.MoveTo(RequiredPosition := StationArray[CurrentStation].EndPosition,
								MoveVelocity := StationArray[CurrentStation].ProcessVelocity,
								NonModuloMove := _NonModuloMoves);
		State := IndexSequenceState.InProcess;
								
	IndexSequenceState.InProcess:
		IF ThisMover.isMoverStationary() THEN 
			IF ThisMover.isMoverAtPosition(StationArray[CurrentStation].EndPosition) THEN
				State := IndexSequenceState.GetNextMove;
			END_IF
		END_IF
	
	IndexSequenceState.GetNextMove:
		IF CurrentStation = SystemParameters.NumberOfStations THEN
			IF ThisMover.MoveTo(RequiredPosition := _startPosition,
							MoveVelocity := _MoverVelocity,
							NonModuloMove := _NonModuloMoves) = 1 THEN
				State := IndexSequenceState.MovingToStart;
				StationArray[CurrentStation].MoverAway();
				CurrentStation := 0; 
			END_IF
		ELSE
			State := IndexSequenceState.GoToNextStation;
		END_IF
		
	IndexSequenceState.GoToNextStation:
		IF StationArray[CurrentStation + 1].IsProcess THEN
			TargetStationPosition := StationArray[CurrentStation + 1].StartPosition;
		ELSE
			TargetStationPosition := StationArray[CurrentStation + 1].Position;
		END_IF
		IF 	ThisMover.MoveTo(RequiredPosition := TargetStationPosition,
							MoveVelocity := _MoverVelocity,
							NonModuloMove := _NonModuloMoves) = 1 THEN
			IF CurrentStation <> 0 THEN
				StationArray[CurrentStation].MoverAway();	
			END_IF		
			CurrentStation := CurrentStation + 1;
			State := IndexSequenceState.MovingToStation;
		END_IF	

	IndexSequenceState.Stopping:
		State := IndexSequenceState.Available;
		CurrentStation := 0;
		TargetStationPosition := 0.0;
	ELSE
		Cycle := E_FAIL;
END_CASE

//Cyclic update info data
stSequenceInfo.CurrentStation := UINT_TO_INT(CurrentStation);
stSequenceInfo.MoverId := ThisMover.AxisRef.NcToPlc.AxisId;
stSequenceInfo.State := State;
stSequenceInfo.Velocity := ThisMover.AxisRef.NcToPlc.ActVelo;
END_METHOD

PROPERTY MoverVelocity : mc_lreal
GET
MoverVelocity := _MoverVelocity;
END_GET
SET
_MoverVelocity := MoverVelocity;
END_SET
END_PROPERTY

PROPERTY MyMover : ITF_XtsMoverAxis
GET
MyMover := ThisMover;
END_GET
SET
ThisMover := MyMover;
END_SET
END_PROPERTY

PROPERTY MyStartPosition : MC_LREAL
GET
MyStartPosition := _startPosition;
END_GET
SET
_startPosition := MyStartPosition;
END_SET
END_PROPERTY

PROPERTY MyStations : ARRAY[1..SystemParameters.NumberOfStations] OF IProcess
GET
MyStations := StationArray;
END_GET
SET
StationArray := MyStations;
END_SET
END_PROPERTY

METHOD StartIndexing : BOOL
VAR_INPUT
END_VAR
ExecuteSequence := true;
END_METHOD

METHOD StopIndexing : BOOL
VAR_INPUT
END_VAR
ExecuteSequence := false;
END_METHOD

PROPERTY XtsNoHome : BOOL
GET
XtsNoHome := _XtsNoHome;
END_GET
SET
_XtsNoHome := XtsNoHome;
END_SET
END_PROPERTY

END_FUNCTION_BLOCK

// ---- Station Class/Process/Process.TcPOU
FUNCTION_BLOCK Process EXTENDS Station IMPLEMENTS IProcess
VAR_INPUT
END_VAR
VAR_OUTPUT
END_VAR
VAR
	_isProcess : BOOL;
	_startPos : MC_LREAL;
	_endPos : MC_LREAL;
	_processVelo : MC_LREAL;
	_TimeInProcess : TIME;
END_VAR

{analysis -2}

METHOD PUBLIC  Cycle : HRESULT
VAR_INPUT
END_VAR
Cycle := SUPER^.Cycle();
END_METHOD

PROPERTY EndPosition : MC_LREAL
GET
EndPosition := _endPos;
END_GET
SET
_endPos := EndPosition;
END_SET
END_PROPERTY

PROPERTY IsProcess : BOOL
GET
IsProcess := _isProcess;
END_GET
SET
_isProcess := IsProcess;
END_SET
END_PROPERTY

PROPERTY ProcessVelocity : MC_LREAL
GET
ProcessVelocity := _processVelo;
END_GET
SET
_processVelo := ProcessVelocity;
END_SET
END_PROPERTY

PROPERTY StartPosition : MC_LREAL
GET
StartPosition := _startPos;
END_GET
SET
_startPos := StartPosition;
END_SET
END_PROPERTY

END_FUNCTION_BLOCK

// ---- Station Class/Station/Station.TcPOU
FUNCTION_BLOCK Station EXTENDS CyclicBase IMPLEMENTS IStation, ICyclic
VAR_INPUT
END_VAR
VAR_OUTPUT
END_VAR
VAR
	_Empty : BOOL;
	_Complete : BOOL;
	_Operating : BOOL;
	_Ready : BOOL;
	_Positions : ARRAY[1..4] OF MC_LREAL := [0.0,0.0,0.0,0.0];
	NumberOfPositions : INT := 0;
	AssignedPositions : INT := 1;
	StationMovers : INT;
	stInfo : stStationInfo;
	_HasMover : BOOL;
	ProductCounter : R_TRIG;
	Products : DINT;
	LastStation : BOOL;
	MyMover : ITF_XtsMoverAxis;
END_VAR

{analysis -2}

METHOD Abort : BOOL
VAR_INPUT
END_VAR
_Complete := FALSE;
_Empty := TRUE;
_Operating := FALSE;
_Ready := TRUE;
Abort := true;
END_METHOD

METHOD PUBLIC  Cycle : HRESULT
VAR_INPUT
END_VAR
//Cyclic info
stInfo.StationPosition := _Positions[1];
stInfo.StationStatus.Empty := _Empty;
stInfo.StationStatus.Complete := _Complete;
stInfo.StationStatus.HasMover := _HasMover;
stInfo.StationStatus.Operating := _Operating;
stInfo.StationStatus.Ready := _Ready;

IF LastStation THEN
	ProductCounter(CLK := _Complete);
	IF ProductCounter.Q THEN
		Products := Products + 1;
	END_IF
END_IF

Cycle := S_OK;
END_METHOD

METHOD HasMover : BOOL
VAR_INPUT
	mover : ITF_XtsMoverAxis;
END_VAR
StationMovers := StationMovers + 1;
IF StationMovers = NumberOfPositions THEN
	_HasMover := TRUE;
END_IF
MyMover := mover;
HasMover := TRUE;
END_METHOD

METHOD IsClear : BOOL
IsClear := _Empty;
END_METHOD

METHOD isComplete : BOOL
isComplete := _Complete;
END_METHOD

PROPERTY PUBLIC IsLastStation : BOOL
GET
IsLastStation := LastStation;
END_GET
SET
LastStation := IsLastStation;
END_SET
END_PROPERTY

METHOD IsOperating : BOOL
IsOperating := _Operating;
END_METHOD

METHOD IsReady : BOOL
IsReady := _Ready;
END_METHOD

METHOD MoverAway : BOOL
VAR_INPUT
END_VAR
StationMovers := StationMovers - 1;
MyMover := 0;
MoverAway := TRUE;
END_METHOD

PROPERTY Position : MC_LREAL
GET
Position := _Positions[AssignedPositions];
AssignedPositions := AssignedPositions + 1;
IF AssignedPositions > NumberOfPositions THEN
	AssignedPositions := 1;
END_IF
END_GET
SET
IF NumberOfPositions < 5 THEN
	NumberOfPositions := NumberOfPositions + 1;
	_Positions[NumberOfPositions] := Position;
END_IF
END_SET
END_PROPERTY

END_FUNCTION_BLOCK

// ---- Station Class/Station/StationSample.TcPOU
FUNCTION_BLOCK StationSample EXTENDS Process
VAR
	_OperationTime : TIME := T#1S;
	Operation : TON;
	State: INT;
END_VAR

{analysis -2}

METHOD Abort : BOOL
VAR_INPUT
END_VAR
SUPER^();

Abort := TRUE;
_Complete := FALSE;
_Empty := TRUE;
_Operating := FALSE;
_Ready := TRUE;
StationMovers := State := 0;
END_METHOD

METHOD Cycle : HRESULT
VAR
	CycleResult : HRESULT;
END_VAR
Cycle := S_OK;
IF _isProcess THEN
	Operation.IN := _HasMover;
	IF NOT Operation.IN THEN
		_TimeInProcess := Operation.ET;
	END_IF
ELSE
	CASE State OF
		0:
			IF _HasMover THEN
				_Operating := TRUE;
				_Empty := FALSE;
				_Ready := FALSE;
				Operation.IN := TRUE;
				State := 1;
			END_IF
		1:
			IF Operation.Q THEN
				_Complete := TRUE;
				IF StationMovers = 0 THEN
					_HasMover := FALSE;
					Operation.IN := FALSE;
				END_IF
				State := 2;
			END_IF
		2:
			_Complete := FALSE;
			_Empty := TRUE;
			_Operating := FALSE;
			_Ready := TRUE;
			State := 0;
		ELSE
			Cycle := E_FAIL;
	END_CASE	
END_IF

Operation(PT := _OperationTime);

CycleResult := SUPER^.Cycle();
stInfo.StationProcessTime := _OperationTime;

IF CycleResult = E_FAIL THEN
	Cycle := E_FAIL;
END_IF
END_METHOD

PROPERTY TempPropTime : time
GET
TempPropTime := _OperationTime;
END_GET
SET
_OperationTime := TempPropTime;
END_SET
END_PROPERTY

END_FUNCTION_BLOCK

// ---- Station Class/TMSStation/TmsEmbarkSingleSwitch.TcPOU
FUNCTION_BLOCK TmsEmbarkSingleSwitch EXTENDS Process IMPLEMENTS ITF_SwitchStation
VAR
	DepartMover : ITF_XtsMoverAxis;
	ExecuteSequence : BOOL;
	SwitchAxis : MC2_Axis_Base;
	_switchLoadPosition : MC_LREAL;
	_switchUnloadPosition : MC_LREAL;
	State :(
		Init,                                               
		Ready,                                 
        Waiting,
		HasSwitch,
		Boarding,
		BoardingComplete,
		Moving,
		ActivateTrackForMover,
		CheckTrackActive,
		ReturnHome,
		Done,
		Aborting); 
	_switchPosition: MC_LREAL;
	_TargetTrackId : I_XtsTrack;
	_BoardVelocity : MC_LREAL;
	_SwitchVelocity : MC_LREAL;
END_VAR

PROPERTY BoardVelocity : MC_LREAL
GET
BoardVelocity := _BoardVelocity;
END_GET
SET
_BoardVelocity := BoardVelocity;
END_SET
END_PROPERTY

METHOD PUBLIC  Cycle : HRESULT
VAR
	ActivateTrackResult : BOOL;
	BoardMoverResult : HRESULT;
	BaseCallResult : HRESULT;
END_VAR
Cycle := S_OK;
CASE State OF
	Init:
		_Operating := _Empty := _Complete := _Ready := _HasMover := FALSE;
		StationMovers := 0;
		State := Ready;
	
	Ready:	
		IF ExecuteSequence THEN
			_Operating := _Complete := _HasMover := FALSE;
			_Empty := _Ready := TRUE;
			StationMovers := 0;
			State := Waiting;
		END_IF
	
	Waiting:
		IF _HasMover THEN
			State := HasSwitch;
			_Operating := TRUE;
			_Empty := FALSE;
			_Ready := FALSE;
			_Complete := FALSE;
		END_IF
	
	HasSwitch:
		IF SwitchAxis.isAtPosition(position := _switchLoadPosition) THEN
			State := Boarding;
		END_IF
			
	Boarding:
		BoardMoverResult := DepartMover.MoveTo(RequiredPosition := _switchPosition, MoveVelocity := _BoardVelocity, NonModuloMove := TRUE);
		IF DepartMover.isMoverAtPosition(position := _switchPosition) THEN
			State := BoardingComplete;
		END_IF
		
	BoardingComplete:
		IF SwitchAxis.MoveToPosition(Position := _switchUnloadPosition, Velocity := _SwitchVelocity) THEN
			State := Moving;
		END_IF
		
	Moving:
		IF NOT SwitchAxis.isStationary() THEN
			State := ActivateTrackForMover;
		END_IF
		
	ActivateTrackForMover:
		DepartMover.ActivateTrack(NewTrack := _TargetTrackId.MyOTCID,Track := _TargetTrackId);		
		State := CheckTrackActive;

	CheckTrackActive:
		IF DepartMover.MoversActiveTrack = _TargetTrackId.MyOTCID AND SwitchAxis.isAtPosition(position := _switchUnloadPosition) THEN
			State := ReturnHome;
			_Complete := TRUE;
		END_IF
	
	ReturnHome:
		IF SwitchAxis.MoveToPosition(Position := _switchLoadPosition, Velocity := _SwitchVelocity) THEN
			State := Done;
		END_IF
			
	Done:
		IF _Complete AND NOT _HasMover THEN
			_Operating := FALSE;
			_Empty := TRUE;
			_Ready := TRUE;
			State := Waiting;
		END_IF

	Aborting:
		State := Ready;	
		DepartMover := 0;
	ELSE
		Cycle := E_FAIL;
END_CASE
BaseCallResult := SUPER^.Cycle();
SwitchAxis.Cycle();
END_METHOD

METHOD DisableLift : HRESULT
VAR_INPUT
END_VAR
SwitchAxis.DisableAxis();
END_METHOD

METHOD EnableLift : HRESULT
VAR_INPUT
END_VAR
SwitchAxis.EnableAxis();
END_METHOD

METHOD HasMover : BOOL
VAR_INPUT
	mover : ITF_XtsMoverAxis;
END_VAR
IF StationMovers <= 2 THEN
	StationMovers := StationMovers + 1;
	DepartMover := mover;
	_HasMover := TRUE;
END_IF
HasMover := TRUE;
END_METHOD

METHOD PUBLIC MoverAway : BOOL
VAR_INPUT
END_VAR
StationMovers := StationMovers - 1;
IF StationMovers = 0 THEN
	_HasMover := FALSE;
END_IF
DepartMover := 0;
MoverAway := TRUE;
END_METHOD

METHOD ResetLift : HRESULT
VAR_INPUT
END_VAR
SwitchAxis.ResetAxis();
END_METHOD

METHOD StartSwitch : BOOL
VAR_INPUT
END_VAR
ExecuteSequence := true;
END_METHOD

METHOD StopSwitch : BOOL
VAR_INPUT
END_VAR
ExecuteSequence := FALSE;
State := Aborting;
END_METHOD

PROPERTY SwitchLoadPosition : MC_LREAL
GET
SwitchLoadPosition := _switchLoadPosition;
END_GET
SET
_switchLoadPosition := SwitchLoadPosition;
END_SET
END_PROPERTY

{warning 'add method implementation '}
METHOD SwitchMoveComplete : BOOL
END_METHOD

PROPERTY SwitchTravelPosition : mc_lreal
GET
SwitchTravelPosition := _switchPosition;
END_GET
SET
_switchPosition := SwitchTravelPosition;
END_SET
END_PROPERTY

PROPERTY SwitchUnloadPosition : MC_LREAL
GET
SwitchUnloadPosition := _switchUnloadPosition;
END_GET
SET
_switchUnloadPosition := SwitchUnloadPosition;
END_SET
END_PROPERTY

PROPERTY SwitchVelocity : MC_LREAL
GET
SwitchVelocity := _SwitchVelocity;
END_GET
SET
_SwitchVelocity := SwitchVelocity;
END_SET
END_PROPERTY

PROPERTY TargetTrackId : I_XtsTrack
GET
TargetTrackId := _TargetTrackId;
END_GET
SET
_TargetTrackId := TargetTrackId;
END_SET
END_PROPERTY

END_FUNCTION_BLOCK

// ---- Station Class/TMSStation/TmsEmbarkStation.TcPOU
FUNCTION_BLOCK TmsEmbarkStation EXTENDS Station IMPLEMENTS ITF_SwitchStation
VAR
	DepartMover : ITF_XtsMoverAxis;
	SwitchAxis : MC2_Axis_Base;
	_switchUpperPosition : MC_LREAL;
	_switchLowerPosition : MC_LREAL;
	ExecuteSequence : BOOL;
	_TrackLevel : INT := 1; //1 is low, 2 is high
	State :(
		Init,                                               
		Ready,                                 
        Waiting,
		HasSwitch,
		Call,
		FindTarget,
		Boarding,
		BoardingComplete,
		ActivateTrackForMover,
		Moving,
		Done,
		Aborting); 
	_switchPosition: MC_LREAL;
	arrTrackIds : ARRAY[1..SystemParameters.NumberOfTracks] OF I_XtsTrack;
	isUpAllowed : BOOL := TRUE;
	isDownAllowed : BOOL := FALSE;
	isMiddleAllowed : BOOL := TRUE;
	_BoardVelocity : MC_LREAL;
	_SwitchVelocity : MC_LREAL;
END_VAR

{analysis -2}

PROPERTY BoardVelocity : MC_LREAL
GET
BoardVelocity := _BoardVelocity;
END_GET
SET
_BoardVelocity := BoardVelocity;
END_SET
END_PROPERTY

METHOD PUBLIC  Cycle : HRESULT
VAR
	ActivateTrackResult : BOOL;
	BoardMoverResult : HRESULT;
	BaseCallResult : HRESULT;
END_VAR
Cycle := S_OK;
CASE State OF
	Init:
		_Operating := _Empty := _Complete := _Ready := _HasMover := FALSE;
		StationMovers := 0;
		State := Ready;
	
	Ready:	
		IF ExecuteSequence THEN
			_Operating := _Complete := _HasMover := FALSE;
			_Empty := _Ready := TRUE;
			StationMovers := 0;
			State := Waiting;
		END_IF
	
	Waiting:
		IF _HasMover THEN
			State := HasSwitch;
			_Operating := TRUE;
			_Empty := FALSE;
			_Ready := FALSE;
			_Complete := FALSE;
		END_IF
	
	HasSwitch:
		IF (_TrackLevel = 1 AND (SwitchAxis.isAtPosition(_switchLowerPosition) ))
			OR (_TrackLevel = 2 AND (SwitchAxis.isAtPosition(_switchUpperPosition))) THEN
					State := Boarding;
		ELSE
			State := Call;
		END_IF	
		
	Call:
		IF SwitchAxis.IsStationary() THEN
			IF _TrackLevel = 1 THEN
				SwitchAxis.MoveToPosition(Position := _switchLowerPosition, Velocity := _SwitchVelocity);
			ELSE
				SwitchAxis.MoveToPosition(Position := _switchUpperPosition, Velocity := _SwitchVelocity);
			END_IF
		ELSE
			State := Waiting;
		END_IF
			
	Boarding:
		BoardMoverResult := DepartMover.MoveTo(RequiredPosition := _switchPosition, MoveVelocity := _BoardVelocity, NonModuloMove := TRUE);
		IF DepartMover.isMoverAtPosition(position := _switchPosition) THEN
			State := BoardingComplete;
		END_IF
		
	BoardingComplete:
		IF _TrackLevel = 1 THEN
			SwitchAxis.MoveToPosition(Position := _switchUpperPosition, Velocity := _SwitchVelocity);
		ELSE
			SwitchAxis.MoveToPosition(Position := _switchLowerPosition, Velocity := _SwitchVelocity);
		END_IF
		State := BoardingComplete;
		
	Moving:
		IF (_TrackLevel = 1 AND SwitchAxis.isAtPosition(position := _switchUpperPosition)) OR
			(_TrackLevel = 2 AND SwitchAxis.isAtPosition(position := _switchLowerPosition)) THEN
			State := ActivateTrackForMover;
		END_IF
		
	ActivateTrackForMover:
		IF _TrackLevel = 1 THEN
			DepartMover.ActivateTrack(NewTrack := arrTrackIds[2].MyOTCID, Track := arrTrackIds[2]);
		ELSE
			DepartMover.ActivateTrack(NewTrack := arrTrackIds[1].MyOTCID, Track := arrTrackIds[1]);
		END_IF
		State := Moving;
		_Complete := TRUE;
			
	Done:
		IF _Complete AND NOT _HasMover THEN
			_Operating := FALSE;
			_Empty := TRUE;
			_Ready := TRUE;
			State := Waiting;
		END_IF	

	Aborting:
		State := Ready;	
		DepartMover := 0;
	ELSE
		Cycle := E_FAIL;
END_CASE
BaseCallResult := SUPER^.Cycle();
SwitchAxis.Cycle();
END_METHOD

METHOD HasMover : BOOL
VAR_INPUT
	mover : ITF_XtsMoverAxis;
END_VAR
IF StationMovers <= 2 THEN
	StationMovers := StationMovers + 1;
	DepartMover := mover;
	_HasMover := TRUE;
END_IF
HasMover := TRUE;
END_METHOD

METHOD PUBLIC MoverAway : BOOL
VAR_INPUT
END_VAR
StationMovers := StationMovers - 1;
IF StationMovers = 0 THEN
	_HasMover := FALSE;
END_IF
DepartMover := 0;
MoverAway := TRUE;
END_METHOD

METHOD StartSwitch : BOOL
VAR_INPUT
END_VAR
ExecuteSequence := TRUE;
END_METHOD

METHOD StopSwitch : BOOL
VAR_INPUT
END_VAR
ExecuteSequence := FALSE;
State := Aborting;
END_METHOD

PROPERTY SwitchLowerPosition : MC_LREAL
GET
END_GET
SET
END_SET
END_PROPERTY

METHOD PUBLIC SwitchMoveComplete : BOOL
VAR_INPUT
END_VAR
_Complete := TRUE;
SwitchMoveComplete := true;
END_METHOD

PROPERTY SwitchTravelPosition : mc_lreal
GET
SwitchTravelPosition := _switchPosition;
END_GET
SET
_switchPosition := SwitchTravelPosition;
END_SET
END_PROPERTY

PROPERTY SwitchUpperPosition : MC_LREAL
GET
END_GET
SET
END_SET
END_PROPERTY

PROPERTY TrackIds : array[1..SystemParameters.NumberOfTracks] of I_XtsTrack
GET
TrackIds := arrTrackIds;
END_GET
SET
arrTrackIds := TrackIds;
END_SET
END_PROPERTY

PROPERTY TrackLevel : INT
GET
TrackLevel := _TrackLevel;
END_GET
SET
_TrackLevel := TrackLevel;
END_SET
END_PROPERTY

END_FUNCTION_BLOCK

// ---- Station Class/TMSStation/TmsHoldStation.TcPOU
FUNCTION_BLOCK TmsHoldStation EXTENDS Process 
VAR
	_EmbarkStation : IStation;
	ExecuteSeqeunce : BOOL;
	HoldMover : ITF_XtsMoverAxis;
	State :(
		Init,                                               
		Ready,                                 
        Waiting,
		Processing,
		Clearing,
		Aborting); 
END_VAR

{analysis -2}

METHOD PUBLIC  Cycle : HRESULT
VAR
	CycleResult : HRESULT;
END_VAR
Cycle := S_OK;
CASE State OF
	Init:
		_Operating := _Empty := _Complete := _Ready := _HasMover := FALSE;
		StationMovers := 0;
		State := Ready;
	
	Ready:	
		IF ExecuteSeqeunce THEN
			_Operating := _Complete := _HasMover := FALSE;
			_Empty := _Ready := TRUE;
			StationMovers := 0;
			State := Waiting;
		END_IF
	
	Waiting:
		IF _HasMover THEN
			State := Processing;
			_Operating := TRUE;
			_Empty := FALSE;
			_Ready := FALSE;
		END_IF
		
	Processing:
		IF _EmbarkStation.IsClear() THEN
			_Complete := TRUE;
			State := Clearing;
		END_IF
		
	Clearing:
		IF NOT _HasMover THEN
			State := Waiting;
			_Operating := FALSE;
			_Empty := TRUE;
			_Ready := TRUE;
			_Complete := FALSE;
			HoldMover := 0;
		END_IF
		
	Aborting:
		State := Ready;
		HoldMover := 0;
		_HasMover := FALSE;
	ELSE
		Cycle := E_FAIL;
END_CASE
CycleResult := SUPER^.Cycle();

IF CycleResult = E_FAIL THEN
	Cycle := E_FAIL;
END_IF
END_METHOD

METHOD HasMover : BOOL
VAR_INPUT
	mover : ITF_XtsMoverAxis;
END_VAR
IF StationMovers <= 2 THEN
	StationMovers := StationMovers + 1;
	HoldMover := mover;
	_HasMover := TRUE;
	HasMover := TRUE;
ELSE
	HasMover := FALSE;
END_IF
END_METHOD

METHOD PUBLIC MoverAway : BOOL
VAR_INPUT
END_VAR
StationMovers := StationMovers - 1;
IF StationMovers = 0 THEN
	_HasMover := FALSE;
END_IF
HoldMover := 0;
MoverAway := TRUE;
END_METHOD

PROPERTY MyEmbarkStation : IStation
GET
MyEmbarkStation := _EmbarkStation;
END_GET
SET
_EmbarkStation := MyEmbarkStation;
END_SET
END_PROPERTY

METHOD StartStation : BOOL
VAR_INPUT
END_VAR
ExecuteSeqeunce := true;
END_METHOD

METHOD StopStation : BOOL
VAR_INPUT
END_VAR
ExecuteSeqeunce := FALSE;
State := Aborting;
END_METHOD

END_FUNCTION_BLOCK

// ---- Tasks/AddMoverToGroupTask.TcPOU
FUNCTION_BLOCK AddMoverToGroupTask EXTENDS TaskBase
VAR_INPUT
END_VAR
VAR_OUTPUT
END_VAR
VAR
	AddtoGrp			: MC_AddAxisToGroup;
	_CaGroup			: ICollisionGroup;
	_Axis				: REFERENCE TO AXIS_REF;
	_addMover : BOOL;
	_moverNumber : UDINT;
END_VAR

{analysis -2}

METHOD Abort : BOOL
AddtoGrp.Execute := FALSE;
Abort := true;
State := 0;
END_METHOD

METHOD AddMover : BOOL
VAR_INPUT
	MoverToAdd : ITF_XtsMoverAxis;
END_VAR
_Axis REF= MoverToAdd.AxisRef;
AddtoGrp.IdentInGroup := MoverToAdd.IdentInGroup;
_Busy := TRUE;
AddMover := _addMover := TRUE;
END_METHOD

METHOD Cycle : HRESULT
VAR_INPUT
END_VAR
Cycle := S_OK;
CASE State OF
	0:
		IF _addMover THEN
			Cycle := S_PENDING;
			_Done := FALSE;
			_Error := FALSE;
			_Busy := TRUE;
			AddtoGrp.Execute := TRUE;
			IF AddtoGrp.Busy THEN
				State := 10;
				_addMover := FALSE;
			END_IF
		END_IF
	
	10:
		IF NOT AddtoGrp.Busy THEN
			IF AddtoGrp.Done THEN
				_Done := TRUE;
			ELSIF AddtoGrp.Error THEN
				_Error := TRUE;
			END_IF
			_Busy := FALSE;
			AddtoGrp.Execute := false;
			State := 0;
			Cycle := S_OK;
		END_IF
	ELSE
		Cycle := E_FAIL;
END_CASE

AddtoGrp(AxesGroup := _CaGroup.GroupRef,
			Axis := _Axis);
END_METHOD

METHOD FB_init : BOOL
VAR_INPUT
	bInitRetains : BOOL; // if TRUE, the retain variables are initialized (warm start / cold start)
	bInCopyCode : BOOL;  // if TRUE, the instance afterwards gets moved into the copy code (online change)
	myCaGroup : ICollisionGroup;	
END_VAR
_CaGroup := myCaGroup;
END_METHOD

END_FUNCTION_BLOCK

// ---- Tasks/DisableGroup.TcPOU
FUNCTION_BLOCK DisableGroup EXTENDS TaskBase
VAR_INPUT
END_VAR
VAR_OUTPUT
END_VAR
VAR
	groupDisable		: MC_GroupDisable;
	_caGroup			: ICollisionGroup;
	_disableGroup : BOOL;
END_VAR

{analysis -2}

METHOD Abort : BOOL
State := 0;
groupDisable.Execute := FALSE;
Abort := true;
END_METHOD

METHOD Cycle : HRESULT
VAR_INPUT
END_VAR
Cycle := S_OK;
CASE State OF
	0:
		IF _disableGroup THEN
			Cycle := S_PENDING;
			_Done := FALSE;
			_Error := FALSE;
			_Busy := TRUE;
			groupDisable.Execute := TRUE;
			IF groupDisable.Busy THEN
				_disableGroup := FALSE;
				State := 10;
				Logger.Send(TC_EVENTS.XtsCaGroupEvents.CAGroupDisabling,'');
			END_IF
		END_IF
	
	10:
		IF NOT groupDisable.Busy THEN
			IF groupDisable.Done THEN
				_Done := TRUE;
				Logger.Send(TC_EVENTS.XtsCaGroupEvents.CAGroupDisabled,'');
			ELSIF groupDisable.Error THEN
				_Error := TRUE;
				Logger.Send(TC_EVENTS.XtsCaGroupEvents.CAGroupDisableError,'');
			END_IF
			_Busy := FALSE;
			groupDisable.Execute := false;
			State := 0;
			Cycle := S_OK;
		END_IF
	ELSE
		Cycle := E_FAIL;
END_CASE


groupDisable(AxesGroup := _caGroup.GroupRef);
END_METHOD

METHOD Execute : BOOL
Execute := _disableGroup := TRUE;
END_METHOD

METHOD FB_init : BOOL
VAR_INPUT
	bInitRetains : BOOL; // if TRUE, the retain variables are initialized (warm start / cold start)
	bInCopyCode : BOOL;  // if TRUE, the instance afterwards gets moved into the copy code (online change)
	MyCaGroup : ICollisionGroup;
END_VAR
_caGroup := MyCaGroup;
END_METHOD

END_FUNCTION_BLOCK

// ---- Tasks/EnableGroup.TcPOU
FUNCTION_BLOCK EnableGroup EXTENDS TaskBase
VAR_INPUT
END_VAR
VAR_OUTPUT
END_VAR
VAR
	groupEnable			: MC_GroupEnable;
	_caGroup			: ICollisionGroup;
	_enableGroup : BOOL;
END_VAR

{analysis -2}

METHOD Abort : BOOL
groupEnable.Execute := FALSE;
Abort := TRUE;
State := 0;
END_METHOD

METHOD Cycle : HRESULT
VAR_INPUT
END_VAR
Cycle := S_OK;
CASE State OF
	0:
		IF _enableGroup THEN
			Cycle := S_PENDING;
			_Done := FALSE;
			_Error := FALSE;
			_Busy := TRUE;
			groupEnable.Execute := TRUE;
			IF groupEnable.Busy THEN
				State := 10;
				_enableGroup := FALSE;
				Logger.Send(TC_EVENTS.XtsCaGroupEvents.CAGroupEnabling,'');
			END_IF
		END_IF
	
	10:
		IF NOT groupEnable.Busy THEN
			IF groupEnable.Done THEN
				_Done := TRUE;
				Logger.Send(TC_EVENTS.XtsCaGroupEvents.CAGroupEnabled,'');
			ELSIF groupEnable.Error THEN
				_Error := TRUE;
				Logger.Send(TC_EVENTS.XtsCaGroupEvents.CAGroupEnableError,'');
			END_IF
			_Busy := FALSE;
			groupEnable.Execute := false;
			State := 0;
			Cycle := S_OK;
		END_IF
	ELSE
		Cycle := E_FAIL;
END_CASE


groupEnable(AxesGroup := _caGroup.GroupRef);
END_METHOD

METHOD Execute : BOOL
Execute := _enableGroup := true;
END_METHOD

METHOD FB_init : BOOL
VAR_INPUT
	bInitRetains : BOOL; // if TRUE, the retain variables are initialized (warm start / cold start)
	bInCopyCode : BOOL;  // if TRUE, the instance afterwards gets moved into the copy code (online change)
	MyCaGroup : ICollisionGroup;	
END_VAR
_caGroup := MyCaGroup;
END_METHOD

END_FUNCTION_BLOCK

// ---- Tasks/RemoveAllMoverFromGroup.TcPOU
FUNCTION_BLOCK RemoveAllMoverFromGroup EXTENDS TaskBase
VAR_INPUT
END_VAR
VAR_OUTPUT
END_VAR
VAR
	RemoveAllFromGrp			: MC_UngroupAllAxes;
	_caGroup			: ICollisionGroup;
	_removeAllMovers : BOOL;
	_errorId: UDINT;
END_VAR

{analysis -2}

METHOD Abort : BOOL
RemoveAllFromGrp.Execute := FALSE;
Abort := true;
State := 0;
END_METHOD

METHOD Cycle : HRESULT
VAR_INPUT
END_VAR
Cycle := S_OK;
CASE State OF
	0:
		IF _removeAllMovers THEN
			Cycle := S_PENDING;
			_Done := FALSE;
			_Error := FALSE;
			_Busy := TRUE;
			RemoveAllFromGrp.Execute := TRUE;
			IF RemoveAllFromGrp.Busy THEN
				_removeAllMovers := FALSE;
				State := 10;
				Logger.Send(TC_EVENTS.XtsCaGroupEvents.CAGroupRemoving,'');
			END_IF
		END_IF
		
	10:
		IF NOT RemoveAllFromGrp.Busy THEN
			IF RemoveAllFromGrp.Done THEN
				_Done := TRUE;
				Logger.Send(TC_EVENTS.XtsCaGroupEvents.AllMoversRemoved,'');
			ELSIF RemoveAllFromGrp.Error THEN
				_Error := TRUE;
				_errorId := RemoveAllFromGrp.ErrorId;
				Logger.Send(TC_EVENTS.XtsCaGroupEvents.CAGroupRemoveError,'');
			END_IF
			_Busy := FALSE;
			RemoveAllFromGrp.Execute := false;
			State := 0;
			Cycle := S_OK;
		END_IF
	ELSE
		Cycle := E_FAIL;
END_CASE


RemoveAllFromGrp(AxesGroup := _caGroup.GroupRef);
END_METHOD

METHOD FB_init : BOOL
VAR_INPUT
	bInitRetains : BOOL; // if TRUE, the retain variables are initialized (warm start / cold start)
	bInCopyCode : BOOL;  // if TRUE, the instance afterwards gets moved into the copy code (online change)
	MyCaGroup : ICollisionGroup;	
END_VAR
_caGroup := MyCaGroup;
END_METHOD

METHOD RemoveAllMover : BOOL
RemoveAllMover := _removeAllMovers := true;
END_METHOD

END_FUNCTION_BLOCK

// ---- Tasks/RemoveMoverFromGroup.TcPOU
FUNCTION_BLOCK RemoveMoverFromGroup EXTENDS TaskBase
VAR
	mcRemoveAxisFromGroup : MC_RemoveAxisFromGroup;
	_GroupRef : ICollisionGroup;
	_Leave: BOOL;
END_VAR

METHOD Cycle : HRESULT
VAR_INPUT
END_VAR
Cycle := S_OK;
CASE State OF
	0:
		IF _Leave THEN
			Cycle := S_PENDING;
			_Done := FALSE;
			_Error := FALSE;
			_Busy := TRUE;
			mcRemoveAxisFromGroup.Execute := TRUE;
			IF mcRemoveAxisFromGroup.Busy THEN
				State := 10;
				_Leave := FALSE;
			END_IF
		END_IF
	
	10:
		IF NOT mcRemoveAxisFromGroup.Busy THEN
			IF mcRemoveAxisFromGroup.Done THEN
				_Done := TRUE;
			ELSIF mcRemoveAxisFromGroup.Error THEN
				_Error := TRUE;
			END_IF
			_Busy := FALSE;
			mcRemoveAxisFromGroup.Execute := FALSE;
			State := 0;
			Cycle := S_OK;
		END_IF
	ELSE
		Cycle := E_FAIL;
END_CASE

mcRemoveAxisFromGroup(AxesGroup := _GroupRef.GroupRef);
END_METHOD

METHOD Execute : BOOL
VAR_INPUT
	AxisID : UDINT;
END_VAR
IF NOT _Leave THEN
	Execute := _Leave := TRUE;
	mcRemoveAxisFromGroup.IdentInGroup := UDINT_TO_IDENTINGROUP(id := AxisID);
ELSE
	Execute := false;
END_IF
END_METHOD

METHOD FB_init : BOOL
VAR_INPUT
	bInitRetains : BOOL; // if TRUE, the retain variables are initialized (warm start / cold start)
	bInCopyCode : BOOL;  // if TRUE, the instance afterwards gets moved into the copy code (online change)
	GroupRef : ICollisionGroup;
END_VAR
_GroupRef := GroupRef;
END_METHOD

END_FUNCTION_BLOCK

// ---- Tasks/ResetGroup.TcPOU
{attribute 'hide_all_locals'}
FUNCTION_BLOCK ResetGroup EXTENDS TaskBase
VAR_INPUT
END_VAR
VAR_OUTPUT
END_VAR
VAR
	groupReset			: MC_GroupReset;
	_caGroup			: ICollisionGroup;
	_resetGroup : BOOL;
END_VAR

{analysis -2}

METHOD Abort : BOOL
groupReset.Execute := FALSE;
State := 0;
Abort := true;
END_METHOD

METHOD Cycle : HRESULT
VAR_INPUT
END_VAR
Cycle := S_OK;
CASE State OF
	0:
		IF _resetGroup THEN
			Cycle := S_PENDING;
			_Done := FALSE;
			_Error := FALSE;
			_Busy := TRUE;
			groupReset.Execute := TRUE;
			IF groupReset.Busy THEN
				State := 10;
				_resetGroup := FALSE;
				Logger.Send(TC_EVENTS.XtsCaGroupEvents.CAGroupResetting,'');
			END_IF
		END_IF
	
	10:
		IF NOT groupReset.Busy THEN
			IF groupReset.Done THEN
				_Done := TRUE;
				Logger.Send(TC_EVENTS.XtsCaGroupEvents.CAGroupResetDone,'');
			ELSIF groupReset.Error THEN
				_Error := TRUE;
				Logger.Send(TC_EVENTS.XtsCaGroupEvents.CAGroupResetError,'');
			END_IF
			_Busy := FALSE;
			groupReset.Execute := false;
			State := 0;
			Cycle := S_OK;
		END_IF
	ELSE
		Cycle := E_FAIL;
END_CASE


groupReset(AxesGroup := _caGroup.GroupRef);
END_METHOD

METHOD Execute : BOOL
Execute := _resetGroup := true;
END_METHOD

METHOD FB_init : BOOL
VAR_INPUT
	bInitRetains : BOOL; // if TRUE, the retain variables are initialized (warm start / cold start)
	bInCopyCode : BOOL;  // if TRUE, the instance afterwards gets moved into the copy code (online change)
	MyCaGroup : ICollisionGroup;	
END_VAR
_caGroup := MyCaGroup;
END_METHOD

END_FUNCTION_BLOCK

// ---- Tasks/StopMoverGroup.TcPOU
FUNCTION_BLOCK StopMoverGroup EXTENDS TaskBase
VAR_INPUT
END_VAR
VAR_OUTPUT
END_VAR
VAR
	groupStop			: MC_GroupStop;
	_caGroup			: ICollisionGroup;
	_stopGroup : BOOL;
	_jerk : MC_LREAL;
	_deceleration : MC_LREAL;
END_VAR

{analysis -2}

METHOD Abort : BOOL
groupStop.Execute := FALSE;
State := 0;
Abort := true;
END_METHOD

METHOD Cycle : HRESULT
VAR_INPUT
END_VAR
Cycle := S_OK;
CASE State OF
	0:
		IF _stopGroup THEN
			Cycle := S_PENDING;
			_Done := FALSE;
			_Error := FALSE;
			_Busy := TRUE;
			groupStop.Execute := TRUE;
			IF groupStop.Busy THEN
				State := 10;
				_stopGroup := FALSE;
				Logger.Send(TC_EVENTS.XtsCaGroupEvents.CAGroupStopping,'');
			END_IF
		END_IF
	10:
		IF groupStop.Done THEN
			_Done := TRUE;
			Logger.Send(TC_EVENTS.XtsCaGroupEvents.CAGroupStopped,'');
		ELSIF groupStop.Error THEN
			_Error := TRUE;
			Logger.Send(TC_EVENTS.XtsCaGroupEvents.CAGroupStopError,'');
		END_IF
		IF _Done OR _Error THEN
			_Busy := FALSE;
			groupStop.Execute := FALSE;
			State := 0;
			Cycle := S_OK;
		END_IF
	ELSE
		Cycle := E_FAIL;
END_CASE


groupStop(AxesGroup := _caGroup.GroupRef);
END_METHOD

PROPERTY PUBLIC Deceleration : MC_LREAL
GET
Deceleration := _deceleration;
END_GET
SET
_deceleration := Deceleration;
END_SET
END_PROPERTY

METHOD Execute : BOOL
_stopGroup := Execute := true;
END_METHOD

METHOD FB_init : BOOL
VAR_INPUT
	bInitRetains : BOOL; // if TRUE, the retain variables are initialized (warm start / cold start)
	bInCopyCode : BOOL;  // if TRUE, the instance afterwards gets moved into the copy code (online change)
	CAGroup : ICollisionGroup;
END_VAR
_caGroup := CAGroup;
END_METHOD

PROPERTY PUBLIC Jerk : MC_LREAL
GET
Jerk := _jerk;
END_GET
SET
_jerk := Jerk;
END_SET
END_PROPERTY

END_FUNCTION_BLOCK

// ---- Tasks/XtsDisableSequence.TcPOU
FUNCTION_BLOCK XtsDisableSequence EXTENDS TaskBase
VAR_INPUT
END_VAR
VAR_OUTPUT
END_VAR
VAR
	_collisionGroup : ICollisionGroup;
	DisableTrigger: BOOL;
	moverNumbers : UINT := 1;
	AllMoversDisabled: BOOL;	
	arrMovers : ARRAY[1..SystemParameters.NumberOfMovers] OF ITF_XtsMoverAxis;
	CaGroupResetResult: BOOL;
END_VAR

{analysis -2}

METHOD Abort : BOOL
VAR
END_VAR
DisableTrigger := FALSE;
State := 0;
Abort := true;
END_METHOD

METHOD Cycle : HRESULT
VAR
	RemoveAllCycleResult : HRESULT;
	GrpStopCycleResult : HRESULT;
	LoggerResult : BOOL;
	CaGroupDisableResult: BOOL;
	DisbleAxisResult: BOOL;
END_VAR
Cycle := S_OK;
CASE State OF
	0:
		IF DisableTrigger THEN
			Cycle := S_PENDING;
			DisableTrigger := FALSE;
			_Busy := TRUE;
			_Done := FALSE;
			_Error := FALSE;
			IF _collisionGroup.GroupState = CAGroupStatus.mcGroupStateMoving THEN
//				FOR moverNumbers := 1 TO SystemParameters.NumberOfMovers DO
//					arrMovers[moverNumbers].HaltAxis();
//				END_FOR
//				LoggerResult := Logger.Send(TC_EVENTS.XtsCaGroupEvents.CAGroupStop,'');
//				State := 10;
				IF _collisionGroup.GroupStop() = 2 THEN
					LoggerResult := Logger.Send(TC_EVENTS.XtsCaGroupEvents.CAGroupStop,'');
					State := 10;
				END_IF
			ELSE
				IF _collisionGroup.RemoveAllMovers() = 2 THEN
					LoggerResult := Logger.Send(TC_EVENTS.XtsCaGroupEvents.CaGroupRemoveMovers,'');
					State := 20;
				END_IF
				
			END_IF
		END_IF
		
	10:
		IF _collisionGroup.GroupState = CAGroupStatus.mcGroupStateStandby THEN
			LoggerResult := Logger.Send(TC_EVENTS.XtsCaGroupEvents.CaGroupRemoveMovers,'');
			IF _collisionGroup.RemoveAllMovers() = 2 THEN
				State := 20;
			END_IF
		END_IF
	
	20:
		IF _collisionGroup.GetAxisCount() = 0 THEN
			FOR moverNumbers := 1 TO SystemParameters.NumberOfMovers DO
				arrMovers[moverNumbers].DisableMover();
			END_FOR
			State := 30;
		END_IF
		
	30:
		AllMoversDisabled := TRUE;
		FOR moverNumbers := 1 TO SystemParameters.NumberOfMovers DO
			AllMoversDisabled := TRUE AND NOT arrMovers[moverNumbers].isMoverEnabled();
		END_FOR
		IF AllMoversDisabled THEN
			LoggerResult := Logger.Send(TC_EVENTS.XtsCaGroupEvents.AllMoversDisabled,'');
			State := 40;
			CaGroupDisableResult := _collisionGroup.Disable();
			LoggerResult := Logger.Send(TC_EVENTS.XtsCaGroupEvents.CAGroupDisable,'');
		END_IF
	40:
		IF _collisionGroup.GroupState = CAGroupStatus.mcGroupStateErrorStop THEN
			CaGroupResetResult := _collisionGroup.Reset();
			LoggerResult := Logger.Send(TC_EVENTS.XtsCaGroupEvents.CAGroupReset,'');
		END_IF	
		State := 50;
		
	50:
		IF _collisionGroup.GroupState = 1 THEN
			State := 0;
			Cycle := S_OK;
			_Busy := FALSE;
			_Done := TRUE;
		END_IF
	ELSE
		Cycle := E_FAIL;
END_CASE



IF RemoveAllCycleResult = E_FAIL OR GrpStopCycleResult = E_FAIL THEN
	Cycle := E_FAIL;
END_IF
END_METHOD

METHOD Disable : BOOL
VAR_INPUT
END_VAR
IF NOT _Busy THEN
	DisableTrigger := Disable := true;
END_IF
END_METHOD

METHOD FB_init : BOOL
VAR_INPUT
	bInitRetains : BOOL; // if TRUE, the retain variables are initialized (warm start / cold start)
	bInCopyCode : BOOL;  // if TRUE, the instance afterwards gets moved into the copy code (online change)
	MyCaGroup : ICollisionGroup;
END_VAR
_collisionGroup := MyCaGroup;
END_METHOD

PROPERTY MoverArray : array[1..SystemParameters.NumberOfMovers] of ITF_XtsMoverAxis
GET
MoverArray := arrMovers;
END_GET
SET
arrMovers := MoverArray;
END_SET
END_PROPERTY

END_FUNCTION_BLOCK

// ---- Tasks/XtsEnableSequence.TcPOU
FUNCTION_BLOCK XtsEnableSequence EXTENDS TaskBase
VAR_INPUT
END_VAR
VAR_OUTPUT
END_VAR
VAR
	_collisionGroup : ICollisionGroup;
	moverNumbers : UINT;
	AllMoversEnabled: BOOL;
	EnableTrigger : BOOL;	
	arrMovers : ARRAY[1..SystemParameters.NumberOfMovers] OF ITF_XtsMoverAxis;
END_VAR

{analysis -2}

METHOD Abort : BOOL
EnableTrigger := FALSE;
State := 0;
END_METHOD

METHOD Cycle : HRESULT
VAR
	CAGroupResetResult : BOOL;
	AddMoverResult : HRESULT;
	AddMoverCallResult : HRESULT;
	EnableMoverResult : BOOL;
	CAGroupEnableResult : BOOL;
	LogSentResult : BOOL;
END_VAR
CASE State OF
	0:
		IF EnableTrigger THEN
			Cycle := S_PENDING;
			State := 10;
			EnableTrigger := FALSE;
			moverNumbers := 1;
			_Busy := TRUE;
			_Done := FALSE;
			_Error := FALSE;
		END_IF
		
	10:
		FOR moverNumbers := 1 TO SystemParameters.NumberOfMovers DO
			arrMovers[moverNumbers].ResetAxis();
		END_FOR
		moverNumbers := 1;
		State := 20;
		
	20:
		IF _collisionGroup.GroupState = CAGroupStatus.mcGroupStateErrorStop THEN
			CAGroupResetResult := _collisionGroup.Reset();
			LogSentResult := Logger.Send(TC_EVENTS.XtsCaGroupEvents.CAGroupReset,'');
		END_IF
		State := 30;
		
	30:
		IF _collisionGroup.AddMoverToThisGroup(MoverToAdd := arrMovers[moverNumbers]) =2 THEN
			LogSentResult := Logger.Send(TC_EVENTS.XtsCaGroupEvents.AddingMoverToGroup,UINT_TO_STRING(moverNumbers));
			State := 40;
		END_IF
		
		
	40:
		IF moverNumbers <> SystemParameters.NumberOfMovers THEN
			moverNumbers := moverNumbers + 1;
			State := 30;
		ELSE
			LogSentResult := Logger.Send(TC_EVENTS.XtsCaGroupEvents.AllMoversAdded,'');
			FOR moverNumbers := 1 TO SystemParameters.NumberOfMovers DO
				arrMovers[moverNumbers].EnableMover();
			END_FOR
			State := 50;
		END_IF
		
	50:
		AllMoversEnabled := TRUE;
		FOR moverNumbers := 1 TO SystemParameters.NumberOfMovers DO
			AllMoversEnabled := TRUE AND arrMovers[moverNumbers].isMoverEnabled();
		END_FOR
		IF AllMoversEnabled THEN
			LogSentResult := Logger.Send(TC_EVENTS.XtsCaGroupEvents.AllMoversEnabled,'');
			CAGroupEnableResult := _collisionGroup.Enable();
			LogSentResult := Logger.Send(TC_EVENTS.XtsCaGroupEvents.CAGroupEnable,'');
			State := 60;
		END_IF
		
	60:
		IF _collisionGroup.GroupState = 2 THEN
			State := 0;
			_Busy := FALSE;
			_Done := TRUE;
			Cycle := S_OK;
		END_IF
	ELSE
		Cycle := E_FAIL;
END_CASE
END_METHOD

METHOD Enable : BOOL
VAR_INPUT
END_VAR
IF NOT _Busy THEN
	EnableTrigger := Enable := true;
END_IF
END_METHOD

METHOD FB_init : BOOL
VAR_INPUT
	bInitRetains : BOOL; // if TRUE, the retain variables are initialized (warm start / cold start)
	bInCopyCode : BOOL;  // if TRUE, the instance afterwards gets moved into the copy code (online change)
	MyCaGroup : ICollisionGroup;
END_VAR
_collisionGroup := MyCaGroup;
END_METHOD

PROPERTY MoverArray : array[1..SystemParameters.NumberOfMovers] of ITF_XtsMoverAxis
GET
MoverArray := arrMovers;
END_GET
SET
arrMovers := MoverArray;
END_SET
END_PROPERTY

END_FUNCTION_BLOCK

// ---- XTS Class/XPU/XTSIOEnvVarWrapper.TcPOU
FUNCTION_BLOCK XTSIOEnvVarWrapper IMPLEMENTS ITF_XTSIOEnvVarWrapper
VAR
	XtsIoEnvironment : Tc3_XTS_Utility.FB_TcIoXtsEnvironment;
	stXtsEnvironmentConfiguration	: ST_XtsEnvironmentConfiguration;
	XPU: Tc3_XTS_Utility.I_TcIoXtsProcessingUnit;
	Initialised : BOOL;
END_VAR

METHOD FB_init : BOOL
VAR_INPUT
	bInitRetains : BOOL; // if TRUE, the retain variables are initialized (warm start / cold start)
	bInCopyCode : BOOL;  // if TRUE, the instance afterwards gets moved into the copy code (online change)
END_VAR
stXtsEnvironmentConfiguration.bEnableInitCaGroup := TRUE;
XtsIoEnvironment.P_XtsEnvironmentConfiguration := stXtsEnvironmentConfiguration;
END_METHOD

METHOD GetCaGroupInterface : I_Mc2CaGroup
VAR_INPUT
	CAGroupNumber : INT;
END_VAR
GetCaGroupInterface := XtsIoEnvironment.Mc2CaGroup(1);
END_METHOD

METHOD PUBLIC GetMotorModuleInterface : I_TcIoXtsPartModule
VAR_INPUT
	PartNumber : INT;
	ModuleNumber : INT;
END_VAR
XPU.PartTcIo(PartNumber).ModuleTcIo(ModuleNumber);
END_METHOD

METHOD PUBLIC GetMoverInterface : I_TcIoXtsXpuMover
VAR_INPUT
	MoverId : INT;
END_VAR
GetMoverInterface := XPU.MoverTcIo(MoverID);
END_METHOD

METHOD PUBLIC GetPartInterface : I_TcIoXtsXpuPart
VAR_INPUT
	PartNumber : INT;
END_VAR
GetPartInterface := XPU.PartTcIo(PartNumber);
END_METHOD

METHOD PUBLIC GetTrackInterface : I_TcIoXtsXpuTrack
VAR_INPUT
	TrackNumber : INT;
END_VAR
GetTrackInterface := XPU.TrackTcIo(TrackNumber);
END_METHOD

METHOD GetXPUInterface : I_TcIoXtsProcessingUnit
VAR_INPUT
END_VAR
GetXPUInterface := XPU;
END_METHOD

METHOD PUBLIC Initialise : BOOL
VAR_INPUT
END_VAR
IF XtsIoEnvironment.Init(TRUE) THEN
	XtsIoEnvironment.Init(FALSE);
	XPU := XtsIoEnvironment.XpuTcIo(1);
	Initialise := Initialised := TRUE;
END_IF
END_METHOD

METHOD IsInitialised : BOOL
VAR_INPUT
END_VAR
IsInitialised := Initialised;
END_METHOD

METHOD IsInSim : BOOL
VAR_INPUT
END_VAR
IF  XPU.GetOperationMode() = OperationMode.Simulation THEN
	IsInSim := TRUE;
END_IF
END_METHOD

METHOD TriggerDetection : BOOL
VAR_INPUT
END_VAR
XPU.TriggerDetection();
TriggerDetection := true;
END_METHOD

METHOD TriggerRedetection : BOOL
VAR_INPUT
END_VAR
TriggerRedetection := XPU.TriggerRedetection();
END_METHOD

END_FUNCTION_BLOCK

// ---- XTS Class/Xts Collision Group/CollisionGroup.TcPOU
FUNCTION_BLOCK CollisionGroup EXTENDS CyclicBase IMPLEMENTS ICollisionGroup, ITF_CAMover
VAR_INPUT
END_VAR
VAR_OUTPUT
END_VAR
VAR
	stGroupInformation : CAGroupInfo;
	_caGroup : Tc3_McCoordinatedMotion.AXES_GROUP_REF;
	_ICaGroup : I_Mc2CaGroup;
	ReadGroupStatus : Tc3_McCoordinatedMotion.MC_GroupReadStatus;
	resetCAGroup : ResetGroup(THIS^);
	enableCAGroup : EnableGroup(THIS^);
	disableCAGroup : DisableGroup(THIS^);
	addMover : AddMoverToGroupTask(THIS^);
	removeAllAxes : RemoveAllMoverFromGroup(THIS^);
	grpStop : StopMoverGroup(THIS^);
	removeMover : RemoveMoverFromGroup(THIS^);
END_VAR

{analysis -2}

METHOD AddMoverToThisGroup : HRESULT
VAR_INPUT
	MoverToAdd : ITF_XtsMoverAxis;
END_VAR
IF NOT addMover.Busy THEN
	addMover.AddMover(MoverToAdd := MoverToAdd);
	MoverToAdd.MyCAGroup  := THIS^;
	AddMoverToThisGroup := 2;
END_IF
END_METHOD

PROPERTY CAGroupXtsIoEnvInterface : I_Mc2CaGroup
GET
CAGroupXtsIoEnvInterface := _ICaGroup;
END_GET
SET
_ICaGroup := CAGroupXtsIoEnvInterface;
END_SET
END_PROPERTY

METHOD Cycle : HRESULT
VAR
	ResetCaGroupResult : HRESULT;
	EnableCaGroupResult : HRESULT;
	DisableCaGroupResult : HRESULT;
	AddMoverCallResult: HRESULT;
	RemoveAllCycleResult: HRESULT;
	GrpStopCycleResult: HRESULT;
END_VAR
IF _ICaGroup <> 0 THEN
	ReadGroupStatus(
	AxesGroup:= _caGroup, 
	Enable:= TRUE );
	ResetCaGroupResult := resetCAGroup.Cycle();
	EnableCaGroupResult := enableCAGroup.Cycle();
	DisableCaGroupResult := disableCAGroup.Cycle();
	AddMoverCallResult := addMover.Cycle();
	RemoveAllCycleResult := removeAllAxes.Cycle();
	GrpStopCycleResult := grpStop.Cycle();
	removeMover.Cycle();
	
	//Cyclic get CaGroup information
	stGroupInformation.sName := 'MainCAGroup';
	stGroupInformation.eGroupState := _caGroup.NcToPlc.Common.GroupStatus.State;
	stGroupInformation.nAxesCount	:= UDINT_TO_INT(_caGroup.NcToPlc.Common.GroupAxesCount);
	stGroupInformation.nId			:= _caGroup.NcToPlc.Common.GroupOID;	
	Cycle := 1;
ELSE
	Cycle := -1;
END_IF
END_METHOD

METHOD Disable : BOOL
VAR_INPUT
END_VAR
IF NOT disableCAGroup.Busy THEN
	disableCAGroup.Execute();
END_IF
END_METHOD

METHOD Enable : BOOL
VAR_INPUT
END_VAR
IF NOT enableCAGroup.Busy THEN
	enableCAGroup.Execute();
END_IF
END_METHOD

METHOD GetAxisCount : udint
VAR_INPUT
END_VAR
GetAxisCount := _caGroup.NcToPlc.Common.GroupAxesCount;
END_METHOD

PROPERTY GroupRef : reference to AXES_GROUP_REF
GET
GroupRef REF= _caGroup;
END_GET
END_PROPERTY

PROPERTY GroupState : CAGroupStatus
GET
IF ReadGroupStatus.GroupDisabled THEN
	GroupState := CAGroupStatus.mcGroupStateDisabled;
ELSIF ReadGroupStatus.GroupErrorStop THEN
	GroupState := CAGroupStatus.mcGroupStateErrorStop;
ELSIF ReadGroupStatus.GroupHoming THEN
	GroupState := CAGroupStatus.mcGroupStateHoming;
ELSIF ReadGroupStatus.GroupMoving THEN
	GroupState := CAGroupStatus.mcGroupStateMoving;
ELSIF ReadGroupStatus.GroupNotReady THEN
	GroupState := CAGroupStatus.mcGroupStateNotReady;
ELSIF ReadGroupStatus.GroupStandby THEN
	GroupState := CAGroupStatus.mcGroupStateStandby;
ELSIF ReadGroupStatus.GroupStopping THEN
	GroupState := CAGroupStatus.mcGroupStateStopping;
ELSIF ReadGroupStatus.Error THEN
	GroupState := CAGroupStatus.mcGroupError;
END_IF
END_GET
END_PROPERTY

METHOD GroupStop : HRESULT
VAR_INPUT
END_VAR
IF NOT grpStop.Busy THEN
	GroupStop := 2;
	grpStop.Execute();
END_IF
END_METHOD

METHOD RemoveAllMovers : HRESULT
VAR_INPUT
END_VAR
IF NOT removeAllAxes.Busy THEN
	removeAllAxes.RemoveAllMover();
	RemoveAllMovers := 2;
END_IF
END_METHOD

METHOD RemoveAMover : BOOL
VAR_INPUT
	moverId : UDINT;
END_VAR
IF NOT removeMover.Busy THEN
	removeMover.Execute(moverid);
END_IF
END_METHOD

METHOD Reset : BOOL
IF NOT resetCAGroup.Busy THEN
	resetCAGroup.Execute();
END_IF
END_METHOD

END_FUNCTION_BLOCK

// ---- XTS Class/Xts Hardware/XTSHardware_V2.TcPOU
FUNCTION_BLOCK XTSHardware_V2 EXTENDS CyclicBase IMPLEMENTS I_Initialise
VAR
	XtsParts : ARRAY[0..SystemParameters.NumberOfParts-1] OF XtsPart;
	XtsTracks : ARRAY[0..SystemParameters.NumberOfTracks-1] OF XtsTrack;
	TrackOTCIDs: ARRAY [1..Tc3_XTS_Utility.TcIoXtsEnvironmentParameterList.MaxXtsTracksPerXpu] OF Tc3_XTS_Utility.OTCID;
	MyXPUInterface : Tc3_XTS_Utility.I_TcIoXtsProcessingUnit;
	MyXtsIoEnvVarRef : ITF_XTSIOEnvVarWrapper;
	XtsIoEnvInitialiseState : INT;
	i: UDINT;
	MyPartCount: UDINT;
	MyTrackCount: UDINT;
	bMoverIdDetectionActive: BOOL;
	bTriggerDetect: BOOL;
	bMoverIdDetectionError: BOOL;
	bMoverIdDetected: BOOL;
END_VAR

METHOD PUBLIC  Cycle : HRESULT
VAR_INPUT
END_VAR
FOR i := 0 TO UDINT_TO_INT(MyPartCount-1) DO
	XtsParts[i].Cycle();
END_FOR
FOR i := 0 TO UDINT_TO_INT(MyTrackCount-1) DO
	XtsTracks[i].Cycle();
END_FOR
END_METHOD

METHOD getAllMoversValid : BOOL
VAR_INPUT
END_VAR
 IF MyXPUInterface.GetAreAllPositionsValid() THEN
	 getAllMoversValid := TRUE;
	 Logger.Send(TC_EVENTS.XtsHardwareEvents.AllMoversValid,'');
 END_IF
END_METHOD

METHOD getMoversDetected : BOOL
VAR_INPUT
END_VAR
IF MyXPUInterface.GetDetectedMoverCount() = MyXPUInterface.GetExpectedMoverCount() THEN
	getMoversDetected := TRUE;
	Logger.Send(TC_EVENTS.XtsHardwareEvents.ExpectedMoversDetected,UDINT_TO_STRING(MyXPUInterface.GetExpectedMoverCount()));
ELSE
	getMoversDetected := FALSE;
	Logger.Send(TC_EVENTS.XtsHardwareEvents.ExpectedMoversNotFound,'');
END_IF
END_METHOD

METHOD GetTrackByOTCID : I_XtsTrack
VAR_INPUT
	trackOTCID : OTCID;
END_VAR
FOR i := 0 TO SystemParameters.NumberOfTracks - 1 DO
	IF trackOTCID = XtsTracks[i].MyOTCID THEN
		GetTrackByOTCID := XtsTracks[i];
	END_IF
END_FOR
END_METHOD

METHOD Initialise : HRESULT
VAR_INPUT
END_VAR

VAR
	
END_VAR
CASE XtsIoEnvInitialiseState OF
	0:
		IF MyXtsIoEnvVarRef <> 0 THEN
			IF MyXtsIoEnvVarRef.IsInitialised() THEN
				MyXPUInterface := MyXtsIoEnvVarRef.GetXPUInterface();
				XtsIoEnvInitialiseState := 1;
			END_IF
		END_IF
	1:
		MyPartCount := MyXPUInterface.GetPartCount();
		IF MyPartCount = SystemParameters.NumberOfParts THEN
			FOR i := 0 TO UDINT_TO_INT(MyPartCount - 1) DO
				XtsParts[i].MyXtsIoEnvInterface := MyXPUInterface.PartTcIo(UDINT_TO_UINT(i + 1));
				IF THIS^.IsInSim() THEN
					XtsParts[i].SetInSim();
				END_IF
			END_FOR
			XtsIoEnvInitialiseState := 3;
		ELSE
			XtsIoEnvInitialiseState := 999;
		END_IF
	3:
		MyTrackCount := MyXPUInterface.GetTrackCount();
		MyXPUInterface.GetTrackOids();
		TrackOTCIDs := MyXPUInterface.P_TrackOids;
		IF MyTrackCount = SystemParameters.NumberOfTracks THEN
			FOR i := 0 TO UDINT_TO_INT(MyTrackCount - 1) DO
				XtsTracks[i].MyXtsIoEnvInterface := MyXPUInterface.TrackTcIo(UDINT_TO_UINT(i + 1));
				XtsTracks[i].MyOTCID := TrackOTCIDs[i + 1];
			END_FOR
			XtsIoEnvInitialiseState := 4;
		ELSE
			XtsIoEnvInitialiseState := 999;
		END_IF
	4:
		XtsIoEnvInitialiseState := 5;
		FOR i := 0 TO UDINT_TO_INT(MyPartCount - 1) DO
			IF XtsParts[i].Initialise() <> 2 THEN
				XtsIoEnvInitialiseState := 4;
			END_IF
		END_FOR
	5:
		XtsIoEnvInitialiseState := 6;
		FOR i := 0 TO UDINT_TO_INT(MyTrackCount - 1) DO
			IF XtsTracks[i].Initialise() <> 2 THEN
				XtsIoEnvInitialiseState := 5;
			END_IF
		END_FOR
	6:
		Initialise := 2;
END_CASE
END_METHOD

METHOD Is24VdcOK : HRESULT
VAR_INPUT
END_VAR
Is24VdcOK := 2;
FOR i := 0 TO (MyXPUInterface.GetPartCount() -1) DO
	IF XtsParts[i].Is24VBusOK() = 1 THEN
		Is24VdcOK := 1;
	END_IF
END_FOR
END_METHOD

METHOD Is48VdcOK : HRESULT
VAR_INPUT
END_VAR
Is48VdcOK := 2;
FOR i := 0 TO (MyXPUInterface.GetPartCount() - 1) DO
	IF XtsParts[i].Is48VBusOK() = 1 THEN
		Is48VdcOK := 1;
	END_IF
END_FOR
END_METHOD

METHOD IsInSim : BOOL
VAR_INPUT
END_VAR
IF  MyXtsIoEnvVarRef.IsInSim() THEN
	IsInSim := TRUE;
	Logger.Send(TC_EVENTS.XtsHardwareEvents.XtsInSimulationMode,'');
ELSE
	IsInSim := FALSE;
END_IF
END_METHOD

PROPERTY MyXtsIoEnvVarWrapper : itf_xtsioenvvarwrapper
GET
MyXtsIoEnvVarWrapper := MyXtsIoEnvVarRef;
END_GET
SET
MyXtsIoEnvVarRef := MyXtsIoEnvVarWrapper;
END_SET
END_PROPERTY

METHOD SetTrackForDetection : BOOL
VAR_INPUT
	TrackToDetect : INT;
END_VAR
IF MyTrackCount = 1 THEN
	MyXPUInterface.TrackTcIo(1).SetIsIncludedInDetection(TRUE);
	Logger.Send(TC_EVENTS.XtsHardwareEvents.ActiveTracksAddedForDetection, UDINT_TO_STRING(MyXPUInterface.GetTrackCount()));
	SetTrackForDetection := TRUE;
ELSE
	IF TrackToDetect <= MyTrackCount THEN 
		SetTrackForDetection := TRUE;
		MyXPUInterface.TrackTcIo(TrackToDetect).SetIsIncludedInDetection(TRUE);
		Logger.Send(TC_EVENTS.XtsHardwareEvents.ActiveTracksAddedForDetection, UDINT_TO_STRING(MyXPUInterface.GetTrackCount()));
	END_IF
END_IF
END_METHOD

METHOD TriggerMoverDetection : BOOL
VAR_INPUT
END_VAR
MyXPUInterface.TriggerRedetection();
Logger.Send(TC_EVENTS.XtsHardwareEvents.MoverDetectionInitiated,'');
TriggerMoverDetection := true;
END_METHOD

METHOD TriggerMoverID : BOOL
VAR_INPUT
END_VAR
// Mover1 Functionality		
// Check if "MoverIdDetectionMode" has been activated under the XtsProcessingUnit object.
IF MyXPUInterface.GetMoverIdDetectionMode() = E_MoverIdDetectionMode.Mover1 THEN

	// Check if the "MoverIdDetection" has already been started or the Mover1 was found.
	IF NOT (bMoverIdDetectionActive OR bMoverIdDetected OR bTriggerDetect) THEN
		
		// Trigger the "MoverIdDetection".
		MyXPUInterface.TriggerMoverIdDetection();
		Logger.Send(TC_EVENTS.XtsHardwareEvents.Mover1DetectionStarted,'');
		bTriggerDetect := true;
	END_IF

	// Check for error or success of "MoverIdDetection".
	bMoverIdDetectionError 	:= MyXPUInterface.GetHasMoverIdDetectionError();
	bMoverIdDetected 	:= MyXPUInterface.GetIsMoverIdDetectionValid();
	bMoverIdDetectionActive	:= MyXPUInterface.GetIsMoverIdDetectionActive();
	
	// If the detection has an error, check for errors in output and try again.
	IF bMoverIdDetectionError THEN
		Logger.Send(TC_EVENTS.XtsHardwareEvents.Mover1DetectionFailed,'');
		RETURN; 
	END_IF

	// Do not process any further until the "MoverId" was deteced.
	IF NOT bMoverIdDetected THEN
		RETURN;
	END_IF	
	TriggerMoverID := TRUE;	
	Logger.Send(TC_EVENTS.XtsHardwareEvents.Mover1DetectionComplete,'');
ELSE
	TriggerMoverID := TRUE;
	Logger.Send(TC_EVENTS.XtsHardwareEvents.StandardMoverNumberingComplete,'');
END_IF
END_METHOD

END_FUNCTION_BLOCK

// ---- XTS Class/Xts Hardware/XtsPart.TcPOU
FUNCTION_BLOCK XtsPart EXTENDS CyclicBase
VAR
	_MyInterface : Tc3_XTS_Utility.I_TcIoXtsXpuPart;
	XtsIoEnvInitialiseState : INT;
	MyModuleCount : UDINT;
	PartDriveState: Tc3_XTS_Utility.DriveState;
	_ReadyToEnable: BOOL;
	MyModules : ARRAY[0..SystemParameters.MaxModulesInPart] OF XtsMotorModule;
	ModuleIndex: UDINT := 1;
	InSim : BOOL;
	i : UINT;
END_VAR

METHOD PUBLIC  Cycle : HRESULT
VAR_INPUT
END_VAR
PartDriveState := _MyInterface.GetDriveState();

CASE PartDriveState OF
	DriveState.Unknown:
		_ReadyToEnable := FALSE;

	DriveState.FaultReactionActive:
		_ReadyToEnable := FALSE;

	DriveState.Fault:
		_ReadyToEnable := FALSE;

	DriveState.NotReadyToSwitchOn:
		_ReadyToEnable := FALSE;

	DriveState.SwitchOnDisabled:
		_ReadyToEnable := FALSE;

	DriveState.ReadyToSwitchOn:
		_ReadyToEnable := TRUE;

	DriveState.SwitchedOn:
		_ReadyToEnable := TRUE;

	DriveState.OperationEnabled:
		_ReadyToEnable := TRUE;

ELSE
	_ReadyToEnable := FALSE;
END_CASE

FOR i := 0 TO (UDINT_TO_UINT(MyModuleCount) - 1) DO
	MyModules[i].Cycle();
END_FOR
END_METHOD

METHOD Initialise : HRESULT
VAR_INPUT
END_VAR
CASE XtsIoEnvInitialiseState OF
	0:
		IF _MyInterface <> 0 THEN
			XtsIoEnvInitialiseState := 1;
		ELSE
			XtsIoEnvInitialiseState := 999;
		END_IF
	1:
		MyModuleCount := _MyInterface.GetModuleCount();
		IF InSim THEN
			XtsIoEnvInitialiseState := 3;
			FOR i := 0 TO UDINT_TO_UINT(MyModuleCount - 1) DO
				MyModules[i].SetInSim();
			END_FOR
			InSim := true;
		ELSE
			FOR i := 0 TO UDINT_TO_UINT(MyModuleCount - 1) DO
				MyModules[i].MyCoEInterface := _MyInterface.ModuleCoE(i + 1);
				MyModules[i].MyModuleInterface := _MyInterface.ModuleTcIo(i + 1);
			END_FOR
			XtsIoEnvInitialiseState := 2;
		END_IF
		
	2:
		XtsIoEnvInitialiseState := 3;
		FOR i := 0 TO UDINT_TO_UINT(MyModuleCount-1) DO
			IF MyModules[i].Initialise() <> 2 THEN
				XtsIoEnvInitialiseState := 2;
			END_IF
		END_FOR
	3:
		Initialise := 2;

END_CASE
END_METHOD

METHOD Is24VBusOK : BOOL
VAR_INPUT
END_VAR
Is24VBusOK := TRUE;
FOR i := 0 TO (UDINT_TO_UINT(MyModuleCount) - 1) DO
	IF MyModules[i].Is24VOK() = 1 THEN
		Is24VBusOK := FALSE;
	END_IF
END_FOR
END_METHOD

METHOD Is48VBusOK : BOOL
VAR_INPUT
END_VAR
Is48VBusOK := TRUE;
FOR i := 0 TO (UDINT_TO_UINT(MyModuleCount) - 1) DO
	IF MyModules[i].Is48VOK() = 1 THEN
		Is48VBusOK := FALSE;
	END_IF
END_FOR
END_METHOD

PROPERTY MyXtsIoEnvInterface : I_TcIoXtsXpuPart
GET
MyXtsIoEnvInterface := _MyInterface;
END_GET
SET
_MyInterface := MyXtsIoEnvInterface;
END_SET
END_PROPERTY

METHOD ResetPart : BOOL
VAR_INPUT
END_VAR
ResetPart := _MyInterface.TriggerReset();
END_METHOD

METHOD SetInSim : HRESULT
VAR_INPUT
END_VAR
InSim := true;
END_METHOD

END_FUNCTION_BLOCK

// ---- XTS Class/Xts Hardware/XtsMotorModule.TcPOU
FUNCTION_BLOCK XtsMotorModule EXTENDS CyclicBase
VAR
	MyModuleIoInterface : I_TcIoXtsPartModule;
	MyModuleCoEInterface : I_AT2xxxXtsMotor;
	CurrentLive: DINT;
	MaxCurrent: DINT;
	Nominal24Vdc : LREAL := 24000;
	Nominal48Vdc : LREAL := 48000;
	InSim : BOOL;
	Module24Vdc: UINT;
	Module48Vdc: UINT;
END_VAR

METHOD PUBLIC  Cycle : HRESULT
VAR_INPUT
END_VAR
IF MyModuleCoEInterface <> 0 AND NOT InSim THEN
	MyModuleCoEInterface.InfoData.Update();
	MyModuleCoEInterface.DiagData.Update();
	//MyModuleCoEInterface.AllCoE.UpdateAllCoEData();
	CurrentLive:=MyModuleCoEInterface.InfoData.OverallCurrent;
	MaxCurrent:=MyModuleCoEInterface.InfoData.MaxOverallCurrentLast500ms;
	Module24Vdc := MyModuleCoEInterface.InfoData.AuxiliaryVoltage24V;
	Module48Vdc := MyModuleCoEInterface.InfoData.DcLinkVoltage;
END_IF
END_METHOD

METHOD Initialise : HRESULT
VAR_INPUT
END_VAR
IF MyModuleIoInterface.P_IsInitialized THEN
	Initialise := 2;
END_IF
END_METHOD

METHOD Is24VOK : HRESULT
VAR_INPUT
END_VAR
IF MyModuleCoEInterface.InfoData.AuxiliaryVoltage24V < (Nominal24Vdc * 0.9) THEN
	Is24VOK := 1;
END_IF
IF MyModuleCoEInterface.InfoData.AuxiliaryVoltage24V > (Nominal24Vdc * 1.1) THEN
	Is24VOK := 1;
END_IF
END_METHOD

METHOD Is48VOK : HRESULT
VAR_INPUT
END_VAR
IF MyModuleCoEInterface.InfoData.DcLinkVoltage < (Nominal48Vdc * 0.9) THEN
	Is48VOK := 1;
END_IF
IF MyModuleCoEInterface.InfoData.DcLinkVoltage > (Nominal48Vdc * 1.1) THEN
	Is48VOK := 1;
END_IF
END_METHOD

PROPERTY MyCoEInterface : I_AT2xxxXtsMotor
GET
MyCoEInterface := MyModuleCoEInterface;
END_GET
SET
MyModuleCoEInterface := MyCoEInterface;
END_SET
END_PROPERTY

PROPERTY MyModuleInterface : I_TcIoXtsPartModule
GET
MyModuleInterface := MyModuleIoInterface;
END_GET
SET
MyModuleIoInterface := MyModuleInterface;
END_SET
END_PROPERTY

METHOD SetInSim : HRESULT
VAR_INPUT
END_VAR
InSim := true;
END_METHOD

END_FUNCTION_BLOCK

// ---- XTS Class/Xts Hardware/XtsTrack.TcPOU
FUNCTION_BLOCK XtsTrack EXTENDS CyclicBase IMPLEMENTS I_XtsTrack
VAR
	_MyInterface : I_TcIoXtsXpuTrack;
	XtsIoEnvInitialiseState : INT;
	MyPartCount : UDINT;
	Parts : REFERENCE TO ARRAY[1..TcIoXtsEnvironmentParameterList.MaxPartsPerTrack] OF ST_PartInfoItems;
	i : INT;
	_TrackLength: LREAL;
	_TrackIsClosed: BOOL;
	_OTCID : OTCID;
END_VAR

METHOD PUBLIC  Cycle : HRESULT
VAR_INPUT
END_VAR
Cycle := 2;
END_METHOD

METHOD Initialise : HRESULT
VAR_INPUT
END_VAR
CASE XtsIoEnvInitialiseState OF
	0:
		IF _MyInterface <> 0 THEN
			XtsIoEnvInitialiseState := 1;
		ELSE
			XtsIoEnvInitialiseState := 999;
		END_IF
	1:
		MyPartCount := _MyInterface.GetPartCount();
		XtsIoEnvInitialiseState := 2;
	2:
		XtsIoEnvInitialiseState := 3;
		Parts REF= _MyInterface.GetPartInfoItems();
		
	3:
		IF _MyInterface.P_IsInitialized THEN
			_TrackLength := _MyInterface.GetLength();
			_TrackIsClosed := _MyInterface.GetIsClosed();
			XtsIoEnvInitialiseState := 4;
		END_IF
	4:
		Initialise := 2;

END_CASE
END_METHOD

PROPERTY MyOTCID : OTCID
GET
MyOTCID := _OTCID;
END_GET
SET
_OTCID := MyOTCID;
END_SET
END_PROPERTY

PROPERTY MyXtsIoEnvInterface : I_TcIoXtsXpuTrack
GET
MyXtsIoEnvInterface := _MyInterface;
END_GET
SET
_MyInterface := MyXtsIoEnvInterface;
END_SET
END_PROPERTY

METHOD RemoveFromDetection : BOOL
VAR_INPUT
END_VAR
RemoveFromDetection := _MyInterface.SetIsIncludedInDetection(False);
END_METHOD

METHOD SetForDetection : BOOL
VAR_INPUT
END_VAR
SetForDetection := _MyInterface.SetIsIncludedInDetection(TRUE);
END_METHOD

PROPERTY TrackLength : MC_Lreal
GET
TrackLength := _MyInterface.GetLength();
END_GET
END_PROPERTY

END_FUNCTION_BLOCK

// ---- XTS Class/Xts.TcPOU
FUNCTION_BLOCK ABSTRACT Xts IMPLEMENTS ICyclic, I_Initialise
VAR
	_homePosition : MC_LREAL;
	_HomeSpeed : MC_LREAL;
	_XtsEnabled : BOOL;
	XtsIoEnvVar : XTSIOEnvVarWrapper;
	mcCollisionGroup : CollisionGroup;
	XtsHardware : XTSHardware_V2 := (MyXtsIoEnvVarWrapper := XtsIoEnvVar);
	XtsHwState : XtsSystemInitialisation;
	EnableSequence : XtsEnableSequence(mcCollisionGroup);
	DisableSequence : XtsDisableSequence(mcCollisionGroup);
	State : UINT;	
	i : UINT;
	AtHome: BOOL;
	_MoverArray : ARRAY[1..SystemParameters.NumberOfMovers] OF ITF_XtsMoverAxis;
	EnabledTrigger : R_TRIG;
	DisabledTrigger : R_TRIG;
END_VAR

{analysis -2}

METHOD PUBLIC ActivateTracksInMovers : BOOL
VAR
	ActivateTrackResult : BOOL;
END_VAR
FOR i := 1 TO SystemParameters.NumberOfMovers DO
	_MoverArray[i].ActivateTrack(newTrack := _MoverArray[i].MoversActiveTrack,
									Track := XtsHardware.GetTrackByOTCID(trackOTCID := _MoverArray[i].MoversActiveTrack));
END_FOR
ActivateTracksInMovers := true;
END_METHOD

METHOD PUBLIC Cycle : HRESULT
VAR
	EnableResult : HRESULT;
	DisableResult : HRESULT;
	GrpStopResult : HRESULT;
	CollisionResult : HRESULT;
END_VAR
EnableResult := EnableSequence.Cycle();
DisableResult := DisableSequence.Cycle();
CollisionResult := mcCollisionGroup.Cycle();
EnabledTrigger(CLK := EnableSequence.Done);
DisabledTrigger(CLK := DisableSequence.Done);
XtsHardware.Cycle();
IF EnabledTrigger.Q THEN
	_XtsEnabled := TRUE;
END_IF
IF DisabledTrigger.Q THEN
	_XtsEnabled := false;
END_IF
IF EnableResult = E_FAIL OR
	DisableResult = E_FAIL OR
	GrpStopResult = E_FAIL OR
	CollisionResult = E_FAIL THEN
	Cycle := E_FAIL;
END_IF
END_METHOD

METHOD DisableXTS : BOOL
VAR_INPUT
END_VAR
DisableXTS := DisableSequence.Disable();
END_METHOD

METHOD EnableXTS : BOOL
VAR_INPUT
END_VAR
EnableSequence.Enable();
END_METHOD

METHOD PUBLIC GetTMSMoverInterface : BOOL
VAR_INPUT
END_VAR
VAR
	//TmsMoverInterface : ITmsMover;
END_VAR
//FOR i := 1 TO SystemParameters.NumberOfMovers DO
//	IF __QUERYINTERFACE(_MoverArray[i],TmsMoverInterface) THEN
//		TmsMoverInterface.SetMoverInterface(MoverInterface := _XtsTrackHardware.GetMoverEnvInterface(i));
//	END_IF
//END_FOR
FOR i := 1 TO SystemParameters.NumberOfMovers DO
	_MoverArray[i].MoverXtsIoEnvInterface := XtsIoEnvVar.GetMoverInterface(i);
END_FOR
END_METHOD

METHOD GetTrackByOCTID : I_XtsTrack
VAR_INPUT
	TrackId : OTCID;
END_VAR
GetTrackByOCTID := XtsHardware.GetTrackByOTCID(trackOTCID := TrackId);
END_METHOD

METHOD Initialise : HRESULT
VAR_INPUT
END_VAR
CASE XtsHwState OF
	XtsSystemInitialisation.Init:
		IF XtsIoEnvVar.Initialise() THEN
			XtsHwState := XtsSystemInitialisation.PassGroupReference;
		END_IF
		
	XtsSystemInitialisation.PassGroupReference:
		mcCollisionGroup.CAGroupXtsIoEnvInterface := XtsIoEnvVar.GetCaGroupInterface(1);
		XtsHwState := XtsSystemInitialisation.InitialiseHardware;
	
	XtsSystemInitialisation.InitialiseHardware:
		IF XtsHardware.Initialise() = 2 THEN
			XtsHwState := XtsSystemInitialisation.SetDetection;
		END_IF
	
	XtsSystemInitialisation.SetDetection:
		IF XtsHardware.SetTrackForDetection(1) THEN
			XtsHwState := XtsSystemInitialisation.Redetect;
		END_IF
		
	XtsSystemInitialisation.Redetect:
		IF XtsHardware.TriggerMoverDetection() THEN
			XtsHwState := XtsSystemInitialisation.MoversValid;
		END_IF
		
	XtsSystemInitialisation.MoversValid:
		IF XtsHardware.getAllMoversValid() THEN
			XtsHwState := XtsSystemInitialisation.AllMoversFound;
		END_IF
	
	XtsSystemInitialisation.AllMoversFound:
		IF XtsHardware.getMoversDetected() THEN
			XtsHwState := XtsSystemInitialisation.XTSMode;
		END_IF
		
	XtsSystemInitialisation.XTSMode:
		IF XtsHardware.IsInSim() THEN
			XtsHwState := XtsSystemInitialisation.MoverIdDetection;
		ELSE
			XtsHwState := XtsSystemInitialisation.CheckModuleVoltages;
		END_IF
		
	XtsSystemInitialisation.CheckModuleVoltages:
		IF XtsHardware.Is24VdcOK() = 2 AND XtsHardware.Is48VdcOK() = 2 THEN
			XtsHwState := XtsSystemInitialisation.MoverIdDetection;
		END_IF
	
	XtsSystemInitialisation.MoverIdDetection:
		IF XtsHardware.TriggerMoverID() THEN
			XtsHwState := XtsSystemInitialisation.HWReady;
			GetTMSMoverInterface();
		END_IF
	
	XtsSystemInitialisation.HWReady:
		Initialise := 2;	
END_CASE
END_METHOD

METHOD IsXtsIdle : BOOL
VAR_INPUT
END_VAR
IsXtsIdle := DisableSequence.Done;
END_METHOD

METHOD IsXtsReady : BOOL
VAR_INPUT
END_VAR
IsXtsReady := _XtsEnabled;
END_METHOD

PROPERTY MoverArray : array[1..SystemParameters.NumberOfMovers] of ITF_XtsMoverAxis
GET
MoverArray := _MoverArray;
END_GET
SET
_MoverArray := MoverArray;
EnableSequence.MoverArray := MoverArray;
DisableSequence.MoverArray := MoverArray;
END_SET
END_PROPERTY

METHOD PUBLIC Abstract MoverHomeSequence : BOOL
VAR_INPUT
END_VAR
END_METHOD

METHOD StopXts : BOOL
VAR_INPUT
END_VAR
mcCollisionGroup.GroupStop();
END_METHOD

END_FUNCTION_BLOCK
